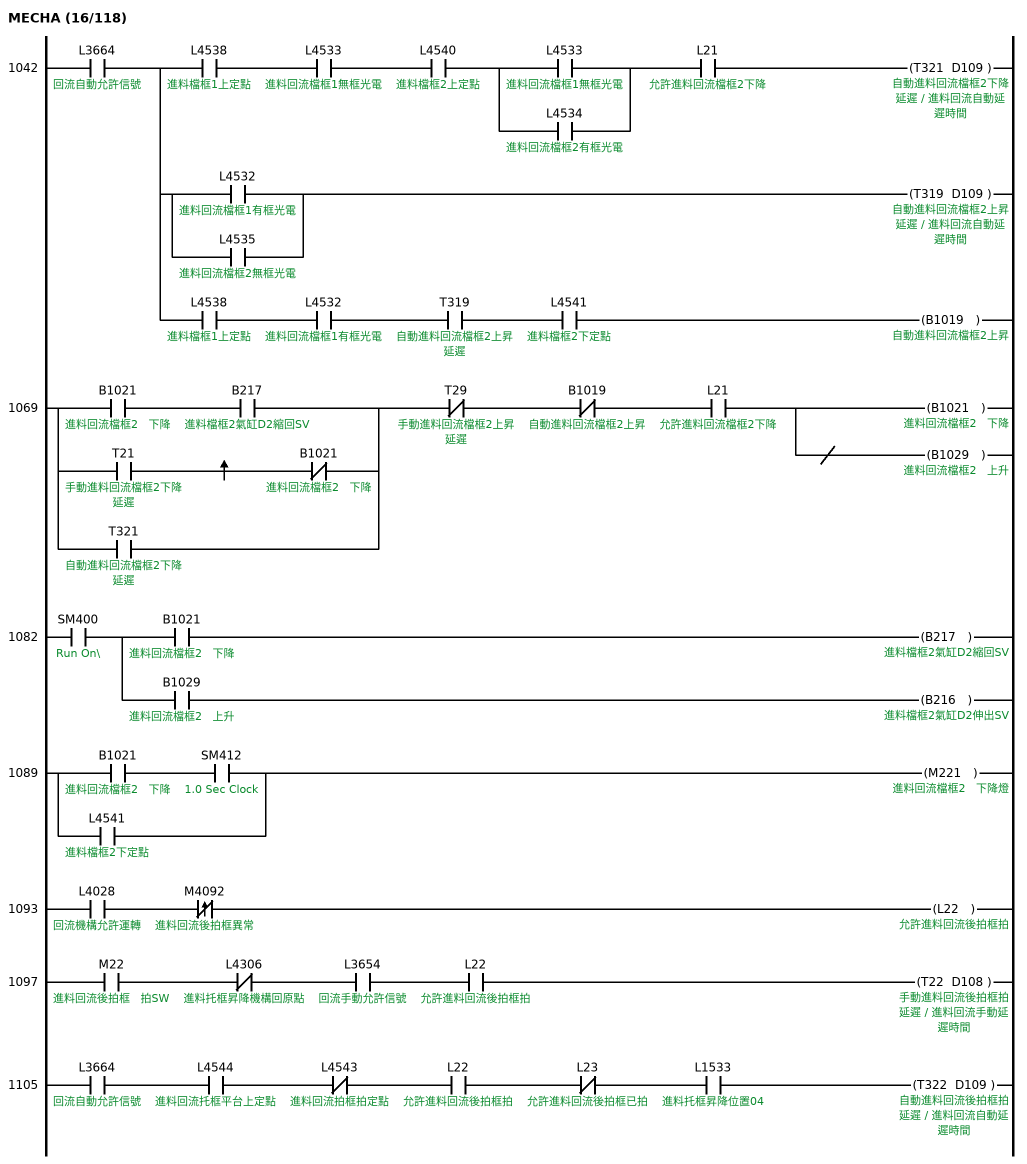
[picture p312: ladder of MECHA, rungs at steps 1042 to 1105]
1042  LD      L3664  ; 回流自動允許信號
      MPS
      AND     L4538  ; 進料檔框1上定點
      AND     L4533  ; 進料回流檔框1無框光電
      AND     L4540  ; 進料檔框2上定點
      LD      L4533  ; 進料回流檔框1無框光電
      OR      L4534  ; 進料回流檔框2有框光電
      ANB
      AND     L21  ; 允許進料回流檔框2下降
      OUT     T321 D109  ; 自動進料回流檔框2下降延遲 / 進料回流自動延遲時間
      MRD
      LD      L4532  ; 進料回流檔框1有框光電
      OR      L4535  ; 進料回流檔框2無框光電
      ANB
      OUT     T319 D109  ; 自動進料回流檔框2上昇延遲 / 進料回流自動延遲時間
      MPP
      AND     L4538  ; 進料檔框1上定點
      AND     L4532  ; 進料回流檔框1有框光電
      AND     T319  ; 自動進料回流檔框2上昇延遲
      AND     L4541  ; 進料檔框2下定點
      OUT     B1019  ; 自動進料回流檔框2上昇
1069  LD      B1021  ; 進料回流檔框2   下降
      AND     B217  ; 進料檔框2氣缸D2縮回SV
      LD      T21  ; 手動進料回流檔框2下降延遲
      MEP
      ANI     B1021  ; 進料回流檔框2   下降
      ORB
      OR      T321  ; 自動進料回流檔框2下降延遲
      ANI     T29  ; 手動進料回流檔框2上昇延遲
      ANI     B1019  ; 自動進料回流檔框2上昇
      AND     L21  ; 允許進料回流檔框2下降
      OUT     B1021  ; 進料回流檔框2   下降
      INV
      OUT     B1029  ; 進料回流檔框2   上升
1082  LD      SM400  ; Run On\
      MPS
      AND     B1021  ; 進料回流檔框2   下降
      OUT     B217  ; 進料檔框2氣缸D2縮回SV
      MPP
      AND     B1029  ; 進料回流檔框2   上升
      OUT     B216  ; 進料檔框2氣缸D2伸出SV
1089  LD      B1021  ; 進料回流檔框2   下降
      AND     SM412  ; 1.0 Sec Clock
      OR      L4541  ; 進料檔框2下定點
      OUT     M221  ; 進料回流檔框2   下降燈
1093  LD      L4028  ; 回流機構允許運轉
      ANDPI   M4092  ; 進料回流後拍框異常
      OUT     L22  ; 允許進料回流後拍框拍
1097  LD      M22  ; 進料回流後拍框   拍SW
      ANI     L4306  ; 進料托框昇降機構回原點
      AND     L3654  ; 回流手動允許信號
      AND     L22  ; 允許進料回流後拍框拍
      OUT     T22 D108  ; 手動進料回流後拍框拍延遲 / 進料回流手動延遲時間
1105  LD      L3664  ; 回流自動允許信號
      AND     L4544  ; 進料回流托框平台上定點
      ANI     L4543  ; 進料回流拍框拍定點
      AND     L22  ; 允許進料回流後拍框拍
      ANI     L23  ; 允許進料回流後拍框已拍
      AND     L1533  ; 進料托框昇降位置04
      OUT     T322 D109  ; 自動進料回流後拍框拍延遲 / 進料回流自動延遲時間
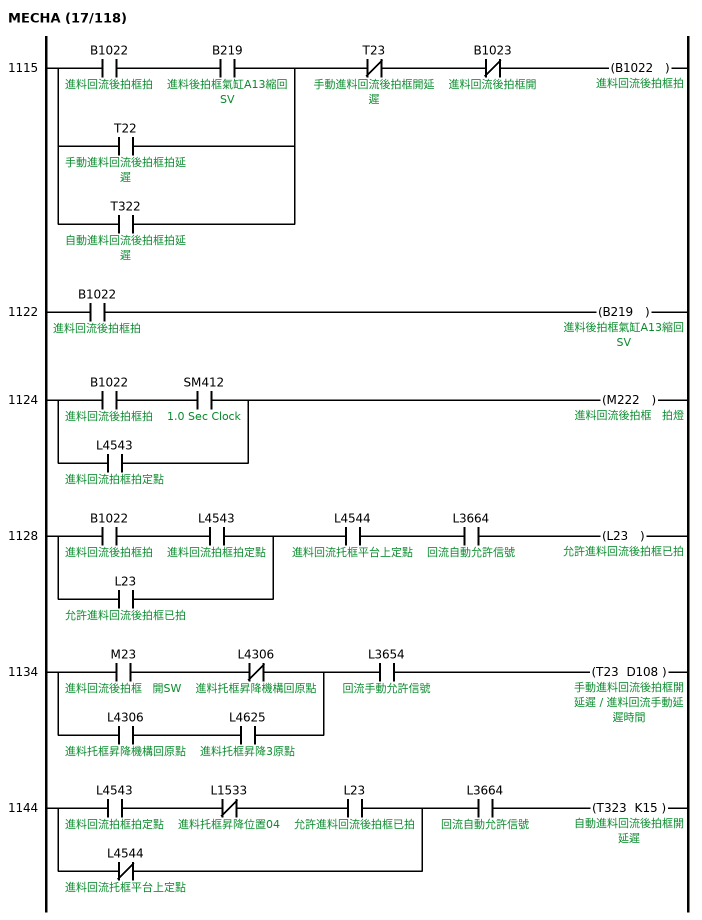
1115  LD      B1022  ; 進料回流後拍框拍
      AND     B219  ; 進料後拍框氣缸A13縮回SV
      OR      T22  ; 手動進料回流後拍框拍延遲
      OR      T322  ; 自動進料回流後拍框拍延遲
      ANI     T23  ; 手動進料回流後拍框開延遲
      ANI     B1023  ; 進料回流後拍框開
      OUT     B1022  ; 進料回流後拍框拍
1122  LD      B1022  ; 進料回流後拍框拍
      OUT     B219  ; 進料後拍框氣缸A13縮回SV
1124  LD      B1022  ; 進料回流後拍框拍
      AND     SM412  ; 1.0 Sec Clock
      OR      L4543  ; 進料回流拍框拍定點
      OUT     M222  ; 進料回流後拍框   拍燈
1128  LD      B1022  ; 進料回流後拍框拍
      AND     L4543  ; 進料回流拍框拍定點
      OR      L23  ; 允許進料回流後拍框已拍
      AND     L4544  ; 進料回流托框平台上定點
      AND     L3664  ; 回流自動允許信號
      OUT     L23  ; 允許進料回流後拍框已拍
1134  LD      M23  ; 進料回流後拍框   開SW
      ANI     L4306  ; 進料托框昇降機構回原點
      LD      L4306  ; 進料托框昇降機構回原點
      AND     L4625  ; 進料托框昇降3原點
      ORB
      AND     L3654  ; 回流手動允許信號
      OUT     T23 D108  ; 手動進料回流後拍框開延遲 / 進料回流手動延遲時間
1144  LD      L4543  ; 進料回流拍框拍定點
      ANI     L1533  ; 進料托框昇降位置04
      AND     L23  ; 允許進料回流後拍框已拍
      ORI     L4544  ; 進料回流托框平台上定點
      AND     L3664  ; 回流自動允許信號
      OUT     T323 K15  ; 自動進料回流後拍框開延遲
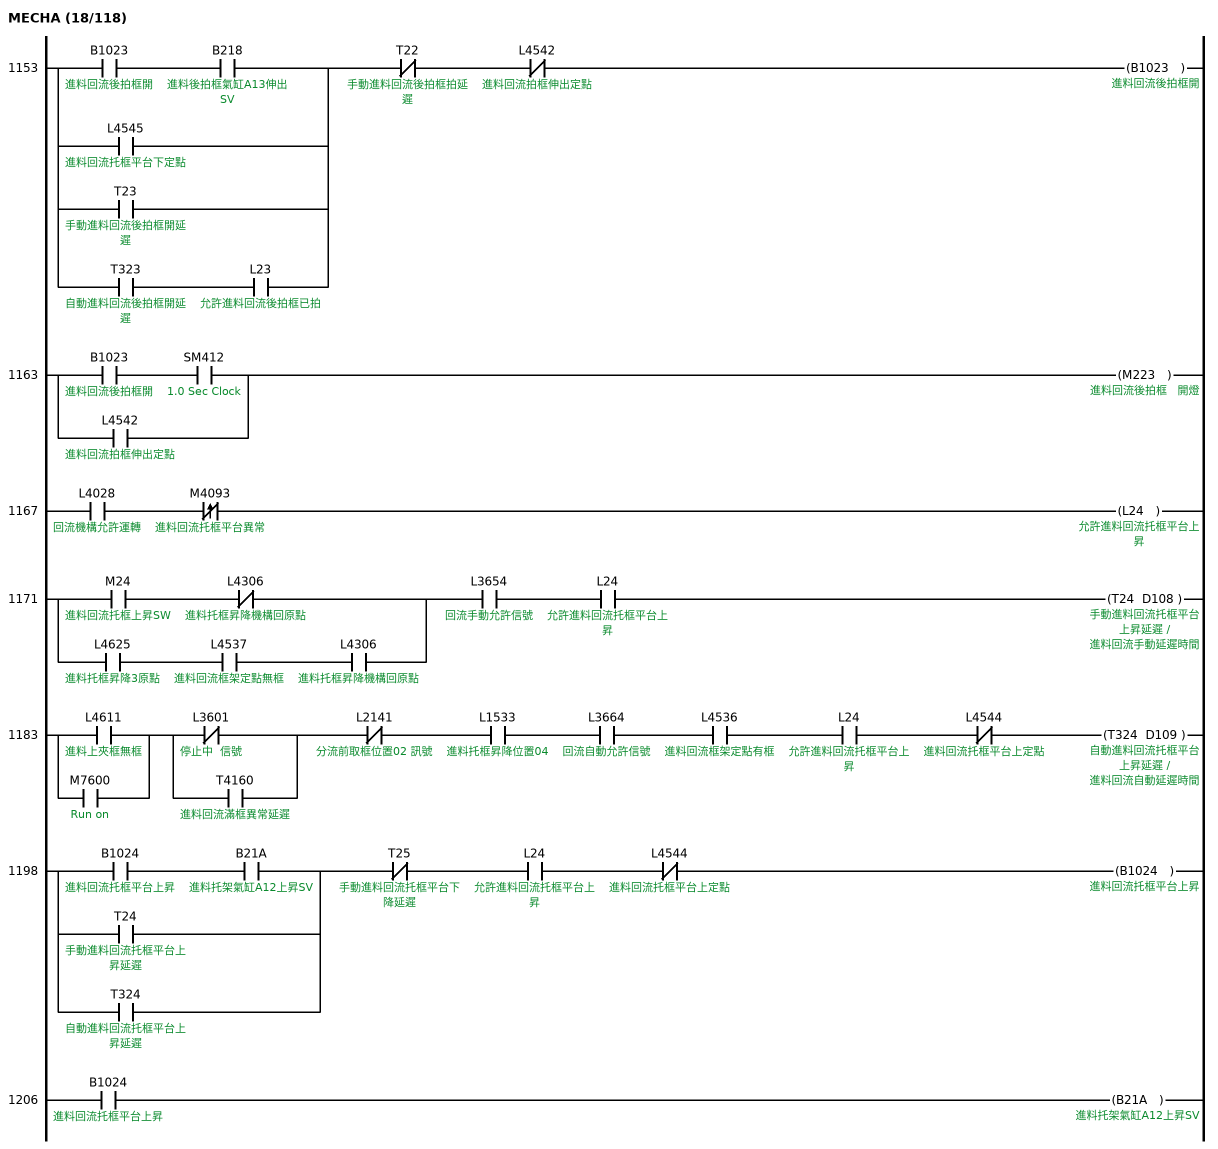
1153  LD      B1023  ; 進料回流後拍框開
      AND     B218  ; 進料後拍框氣缸A13伸出SV
      OR      L4545  ; 進料回流托框平台下定點
      OR      T23  ; 手動進料回流後拍框開延遲
      LD      T323  ; 自動進料回流後拍框開延遲
      AND     L23  ; 允許進料回流後拍框已拍
      ORB
      ANI     T22  ; 手動進料回流後拍框拍延遲
      ANI     L4542  ; 進料回流拍框伸出定點
      OUT     B1023  ; 進料回流後拍框開
1163  LD      B1023  ; 進料回流後拍框開
      AND     SM412  ; 1.0 Sec Clock
      OR      L4542  ; 進料回流拍框伸出定點
      OUT     M223  ; 進料回流後拍框   開燈
1167  LD      L4028  ; 回流機構允許運轉
      ANDPI   M4093  ; 進料回流托框平台異常
      OUT     L24  ; 允許進料回流托框平台上昇
1171  LD      M24  ; 進料回流托框上昇SW
      ANI     L4306  ; 進料托框昇降機構回原點
      LD      L4625  ; 進料托框昇降3原點
      AND     L4537  ; 進料回流框架定點無框
      AND     L4306  ; 進料托框昇降機構回原點
      ORB
      AND     L3654  ; 回流手動允許信號
      AND     L24  ; 允許進料回流托框平台上昇
      OUT     T24 D108  ; 手動進料回流托框平台上昇延遲 / 進料回流手動延遲時間
1183  LD      L4611  ; 進料上夾框無框
      OR      M7600  ; Run on
      LDI     L3601  ; 停止中  信號
      OR      T4160  ; 進料回流滿框異常延遲
      ANB
      ANI     L2141  ; 分流前取框位置02 訊號
      AND     L1533  ; 進料托框昇降位置04
      AND     L3664  ; 回流自動允許信號
      AND     L4536  ; 進料回流框架定點有框
      AND     L24  ; 允許進料回流托框平台上昇
      ANI     L4544  ; 進料回流托框平台上定點
      OUT     T324 D109  ; 自動進料回流托框平台上昇延遲 / 進料回流自動延遲時間
1198  LD      B1024  ; 進料回流托框平台上昇
      AND     B21A  ; 進料托架氣缸A12上昇SV
      OR      T24  ; 手動進料回流托框平台上昇延遲
      OR      T324  ; 自動進料回流托框平台上昇延遲
      ANI     T25  ; 手動進料回流托框平台下降延遲
      AND     L24  ; 允許進料回流托框平台上昇
      ANI     L4544  ; 進料回流托框平台上定點
      OUT     B1024  ; 進料回流托框平台上昇
1206  LD      B1024  ; 進料回流托框平台上昇
      OUT     B21A  ; 進料托架氣缸A12上昇SV
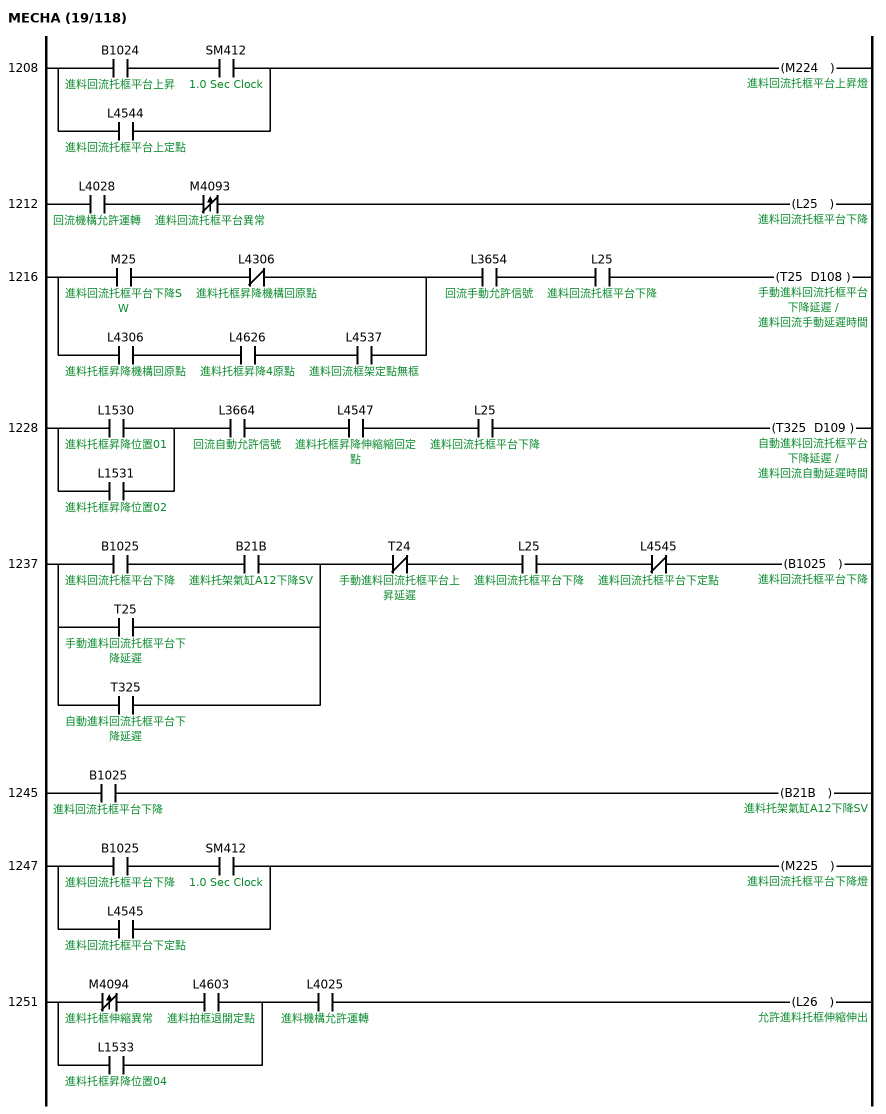
1208  LD      B1024  ; 進料回流托框平台上昇
      AND     SM412  ; 1.0 Sec Clock
      OR      L4544  ; 進料回流托框平台上定點
      OUT     M224  ; 進料回流托框平台上昇燈
1212  LD      L4028  ; 回流機構允許運轉
      ANDPI   M4093  ; 進料回流托框平台異常
      OUT     L25  ; 進料回流托框平台下降
1216  LD      M25  ; 進料回流托框平台下降SW
      ANI     L4306  ; 進料托框昇降機構回原點
      LD      L4306  ; 進料托框昇降機構回原點
      AND     L4626  ; 進料托框昇降4原點
      AND     L4537  ; 進料回流框架定點無框
      ORB
      AND     L3654  ; 回流手動允許信號
      AND     L25  ; 進料回流托框平台下降
      OUT     T25 D108  ; 手動進料回流托框平台下降延遲 / 進料回流手動延遲時間
1228  LD      L1530  ; 進料托框昇降位置01
      OR      L1531  ; 進料托框昇降位置02
      AND     L3664  ; 回流自動允許信號
      AND     L4547  ; 進料托框昇降伸縮縮回定點
      AND     L25  ; 進料回流托框平台下降
      OUT     T325 D109  ; 自動進料回流托框平台下降延遲 / 進料回流自動延遲時間
1237  LD      B1025  ; 進料回流托框平台下降
      AND     B21B  ; 進料托架氣缸A12下降SV
      OR      T25  ; 手動進料回流托框平台下降延遲
      OR      T325  ; 自動進料回流托框平台下降延遲
      ANI     T24  ; 手動進料回流托框平台上昇延遲
      AND     L25  ; 進料回流托框平台下降
      ANI     L4545  ; 進料回流托框平台下定點
      OUT     B1025  ; 進料回流托框平台下降
1245  LD      B1025  ; 進料回流托框平台下降
      OUT     B21B  ; 進料托架氣缸A12下降SV
1247  LD      B1025  ; 進料回流托框平台下降
      AND     SM412  ; 1.0 Sec Clock
      OR      L4545  ; 進料回流托框平台下定點
      OUT     M225  ; 進料回流托框平台下降燈
1251  LDPI    M4094  ; 進料托框伸縮異常
      AND     L4603  ; 進料拍框退開定點
      OR      L1533  ; 進料托框昇降位置04
      AND     L4025  ; 進料機構允許運轉
      OUT     L26  ; 允許進料托框伸縮伸出
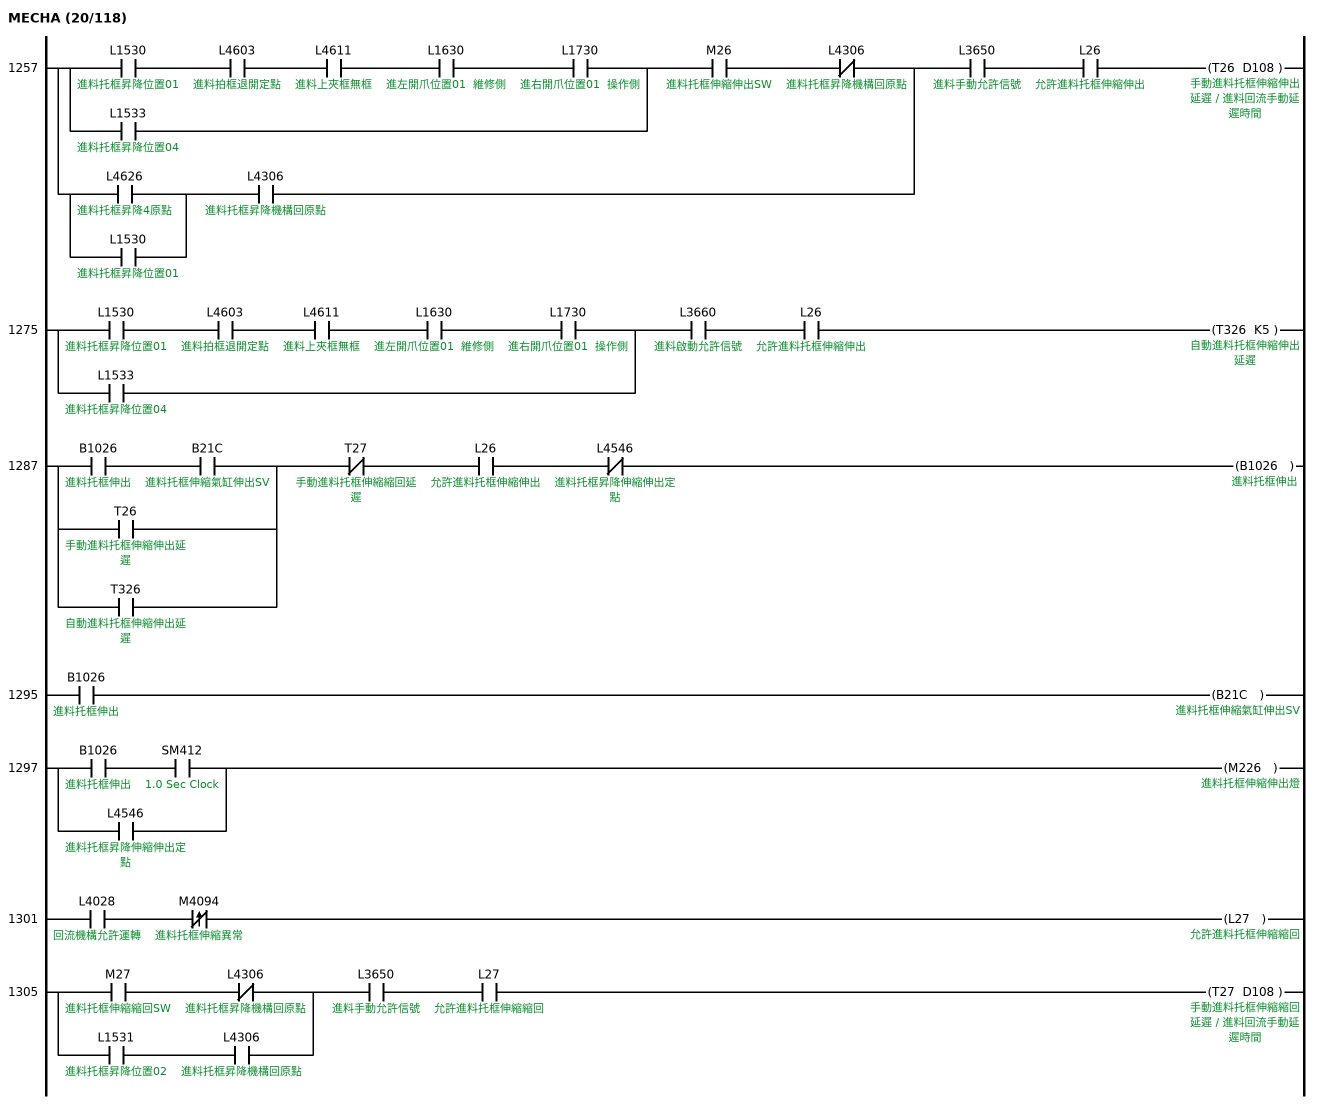
1257  LD      L1530  ; 進料托框昇降位置01
      AND     L4603  ; 進料拍框退開定點
      AND     L4611  ; 進料上夾框無框
      AND     L1630  ; 進左開爪位置01  維修側
      AND     L1730  ; 進右開爪位置01  操作側
      OR      L1533  ; 進料托框昇降位置04
      AND     M26  ; 進料托框伸縮伸出SW
      ANI     L4306  ; 進料托框昇降機構回原點
      LD      L4626  ; 進料托框昇降4原點
      OR      L1530  ; 進料托框昇降位置01
      AND     L4306  ; 進料托框昇降機構回原點
      ORB
      AND     L3650  ; 進料手動允許信號
      AND     L26  ; 允許進料托框伸縮伸出
      OUT     T26 D108  ; 手動進料托框伸縮伸出延遲 / 進料回流手動延遲時間
1275  LD      L1530  ; 進料托框昇降位置01
      AND     L4603  ; 進料拍框退開定點
      AND     L4611  ; 進料上夾框無框
      AND     L1630  ; 進左開爪位置01  維修側
      AND     L1730  ; 進右開爪位置01  操作側
      OR      L1533  ; 進料托框昇降位置04
      AND     L3660  ; 進料啟動允許信號
      AND     L26  ; 允許進料托框伸縮伸出
      OUT     T326 K5  ; 自動進料托框伸縮伸出延遲
1287  LD      B1026  ; 進料托框伸出
      AND     B21C  ; 進料托框伸縮氣缸伸出SV
      OR      T26  ; 手動進料托框伸縮伸出延遲
      OR      T326  ; 自動進料托框伸縮伸出延遲
      ANI     T27  ; 手動進料托框伸縮縮回延遲
      AND     L26  ; 允許進料托框伸縮伸出
      ANI     L4546  ; 進料托框昇降伸縮伸出定點
      OUT     B1026  ; 進料托框伸出
1295  LD      B1026  ; 進料托框伸出
      OUT     B21C  ; 進料托框伸縮氣缸伸出SV
1297  LD      B1026  ; 進料托框伸出
      AND     SM412  ; 1.0 Sec Clock
      OR      L4546  ; 進料托框昇降伸縮伸出定點
      OUT     M226  ; 進料托框伸縮伸出燈
1301  LD      L4028  ; 回流機構允許運轉
      ANDPI   M4094  ; 進料托框伸縮異常
      OUT     L27  ; 允許進料托框伸縮縮回
1305  LD      M27  ; 進料托框伸縮縮回SW
      ANI     L4306  ; 進料托框昇降機構回原點
      LD      L1531  ; 進料托框昇降位置02
      AND     L4306  ; 進料托框昇降機構回原點
      ORB
      AND     L3650  ; 進料手動允許信號
      AND     L27  ; 允許進料托框伸縮縮回
      OUT     T27 D108  ; 手動進料托框伸縮縮回延遲 / 進料回流手動延遲時間
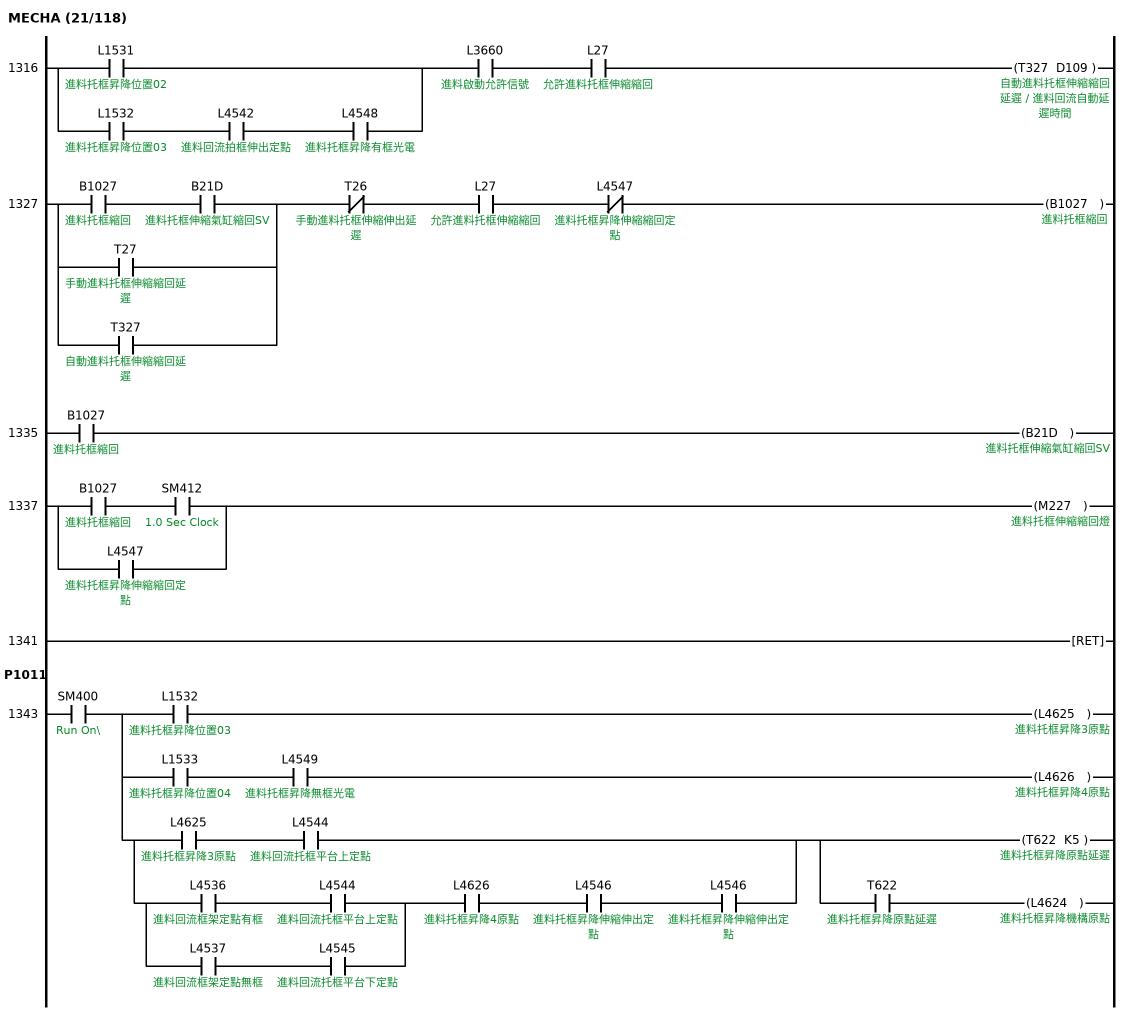
1316  LD      L1531  ; 進料托框昇降位置02
      LD      L1532  ; 進料托框昇降位置03
      AND     L4542  ; 進料回流拍框伸出定點
      AND     L4548  ; 進料托框昇降有框光電
      ORB
      AND     L3660  ; 進料啟動允許信號
      AND     L27  ; 允許進料托框伸縮縮回
      OUT     T327 D109  ; 自動進料托框伸縮縮回延遲 / 進料回流自動延遲時間
1327  LD      B1027  ; 進料托框縮回
      AND     B21D  ; 進料托框伸縮氣缸縮回SV
      OR      T27  ; 手動進料托框伸縮縮回延遲
      OR      T327  ; 自動進料托框伸縮縮回延遲
      ANI     T26  ; 手動進料托框伸縮伸出延遲
      AND     L27  ; 允許進料托框伸縮縮回
      ANI     L4547  ; 進料托框昇降伸縮縮回定點
      OUT     B1027  ; 進料托框縮回
1335  LD      B1027  ; 進料托框縮回
      OUT     B21D  ; 進料托框伸縮氣缸縮回SV
1337  LD      B1027  ; 進料托框縮回
      AND     SM412  ; 1.0 Sec Clock
      OR      L4547  ; 進料托框昇降伸縮縮回定點
      OUT     M227  ; 進料托框伸縮縮回燈
1341  RET
      P1011
1343  LD      SM400  ; Run On\
      MPS
      AND     L1532  ; 進料托框昇降位置03
      OUT     L4625  ; 進料托框昇降3原點
      MRD
      AND     L1533  ; 進料托框昇降位置04
      AND     L4549  ; 進料托框昇降無框光電
      OUT     L4626  ; 進料托框昇降4原點
      MPP
      LD      L4625  ; 進料托框昇降3原點
      AND     L4544  ; 進料回流托框平台上定點
      LD      L4536  ; 進料回流框架定點有框
      AND     L4544  ; 進料回流托框平台上定點
      LD      L4537  ; 進料回流框架定點無框
      AND     L4545  ; 進料回流托框平台下定點
      ORB
      AND     L4626  ; 進料托框昇降4原點
      AND     L4546  ; 進料托框昇降伸縮伸出定點
      AND     L4546  ; 進料托框昇降伸縮伸出定點
      ORB
      ANB
      OUT     T622 K5  ; 進料托框昇降原點延遲
      AND     T622  ; 進料托框昇降原點延遲
      OUT     L4624  ; 進料托框昇降機構原點
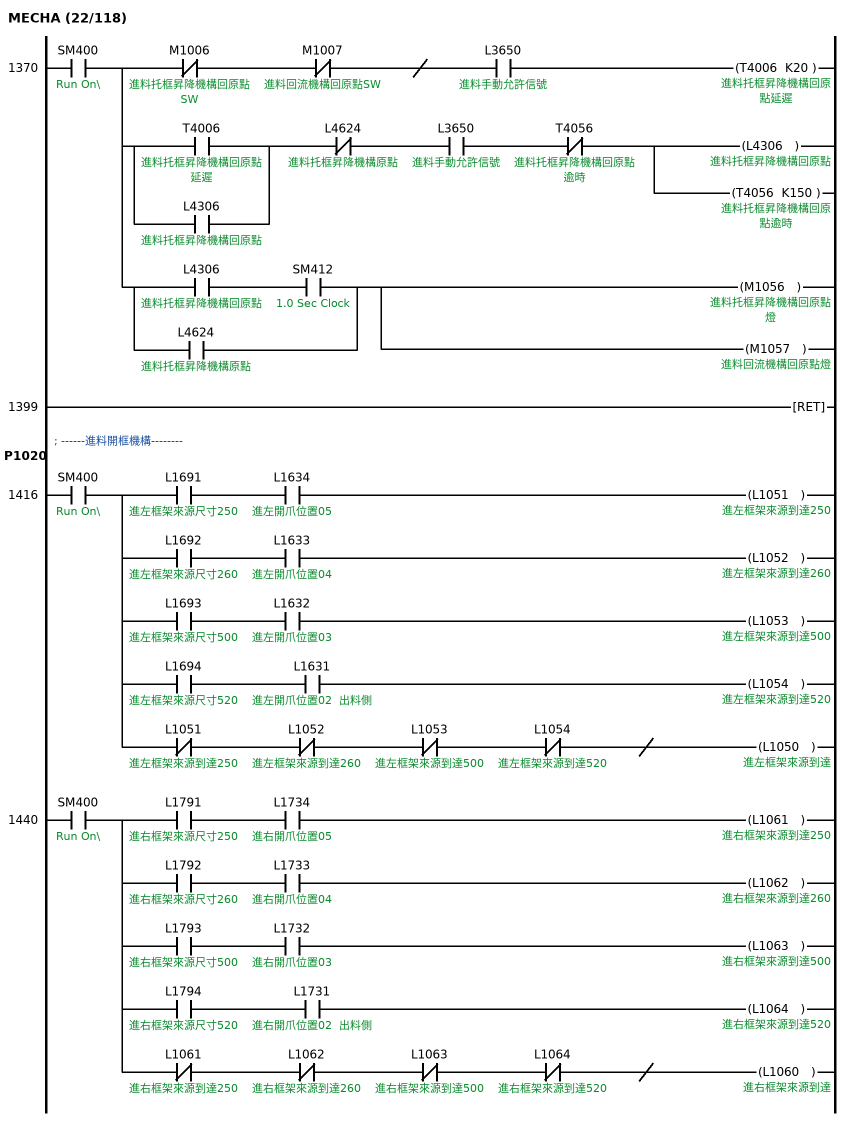
1370  LD      SM400  ; Run On\
      MPS
      ANI     M1006  ; 進料托框昇降機構回原點SW
      ANI     M1007  ; 進料回流機構回原點SW
      INV
      AND     L3650  ; 進料手動允許信號
      OUT     T4006 K20  ; 進料托框昇降機構回原點延遲
      MRD
      LD      T4006  ; 進料托框昇降機構回原點延遲
      OR      L4306  ; 進料托框昇降機構回原點
      ANB
      ANI     L4624  ; 進料托框昇降機構原點
      AND     L3650  ; 進料手動允許信號
      ANI     T4056  ; 進料托框昇降機構回原點逾時
      OUT     L4306  ; 進料托框昇降機構回原點
      OUT     T4056 K150  ; 進料托框昇降機構回原點逾時
      MPP
      LD      L4306  ; 進料托框昇降機構回原點
      AND     SM412  ; 1.0 Sec Clock
      OR      L4624  ; 進料托框昇降機構原點
      ANB
      OUT     M1056  ; 進料托框昇降機構回原點燈
      OUT     M1057  ; 進料回流機構回原點燈
1399  RET
; ------進料開框機構--------
      P1020
1416  LD      SM400  ; Run On\
      MPS
      AND     L1691  ; 進左框架來源尺寸250
      AND     L1634  ; 進左開爪位置05
      OUT     L1051  ; 進左框架來源到達250
      MRD
      AND     L1692  ; 進左框架來源尺寸260
      AND     L1633  ; 進左開爪位置04
      OUT     L1052  ; 進左框架來源到達260
      MRD
      AND     L1693  ; 進左框架來源尺寸500
      AND     L1632  ; 進左開爪位置03
      OUT     L1053  ; 進左框架來源到達500
      MRD
      AND     L1694  ; 進左框架來源尺寸520
      AND     L1631  ; 進左開爪位置02  出料側
      OUT     L1054  ; 進左框架來源到達520
      MPP
      ANI     L1051  ; 進左框架來源到達250
      ANI     L1052  ; 進左框架來源到達260
      ANI     L1053  ; 進左框架來源到達500
      ANI     L1054  ; 進左框架來源到達520
      INV
      OUT     L1050  ; 進左框架來源到達
1440  LD      SM400  ; Run On\
      MPS
      AND     L1791  ; 進右框架來源尺寸250
      AND     L1734  ; 進右開爪位置05
      OUT     L1061  ; 進右框架來源到達250
      MRD
      AND     L1792  ; 進右框架來源尺寸260
      AND     L1733  ; 進右開爪位置04
      OUT     L1062  ; 進右框架來源到達260
      MRD
      AND     L1793  ; 進右框架來源尺寸500
      AND     L1732  ; 進右開爪位置03
      OUT     L1063  ; 進右框架來源到達500
      MRD
      AND     L1794  ; 進右框架來源尺寸520
      AND     L1731  ; 進右開爪位置02  出料側
      OUT     L1064  ; 進右框架來源到達520
      MPP
      ANI     L1061  ; 進右框架來源到達250
      ANI     L1062  ; 進右框架來源到達260
      ANI     L1063  ; 進右框架來源到達500
      ANI     L1064  ; 進右框架來源到達520
      INV
      OUT     L1060  ; 進右框架來源到達
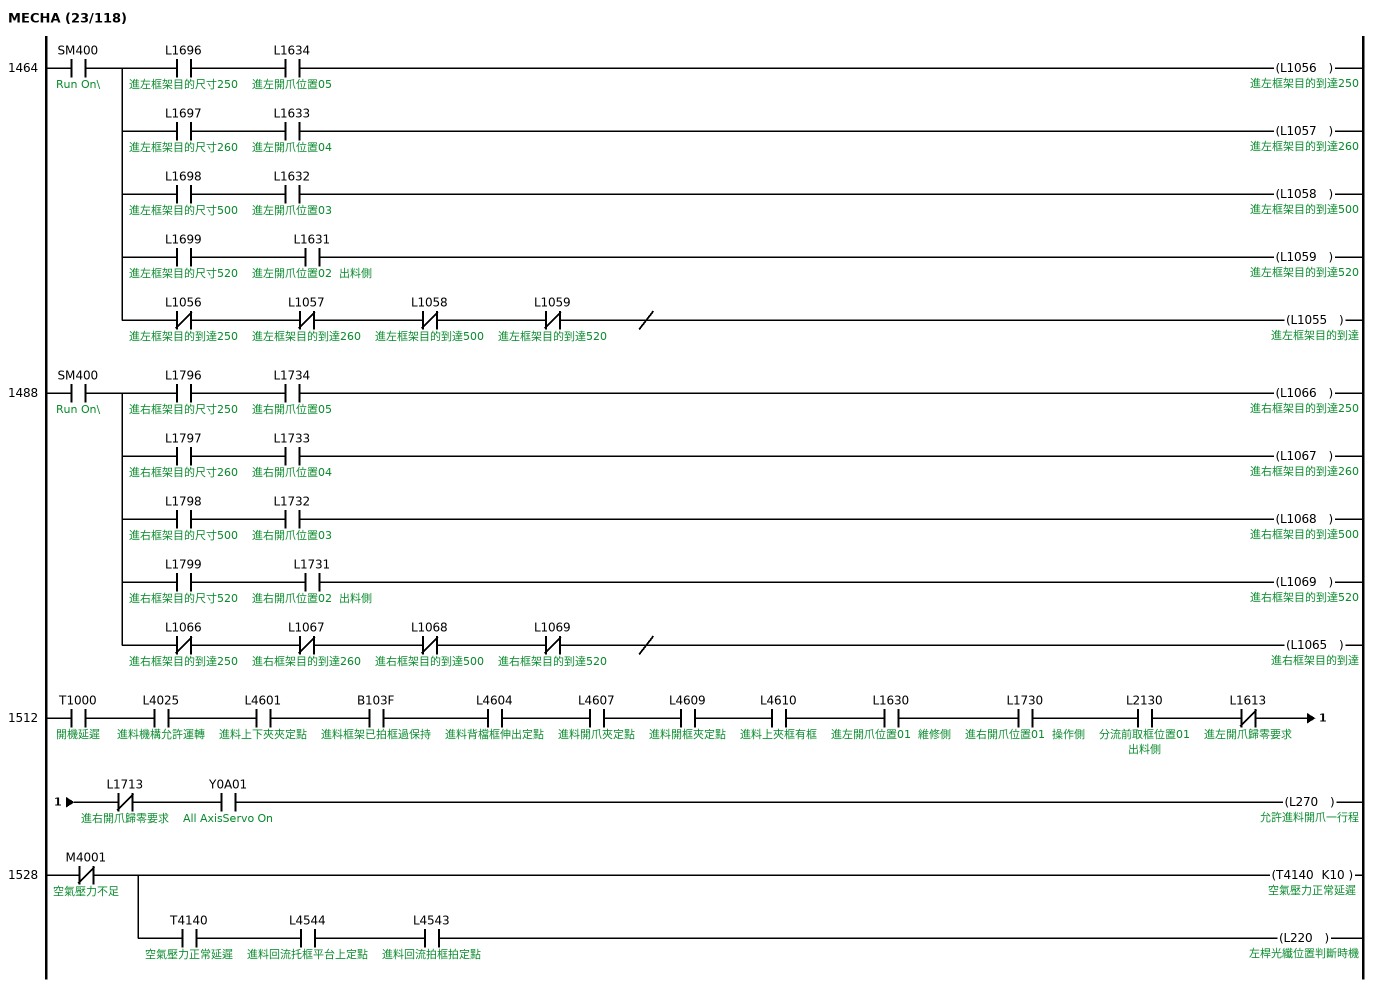
1464  LD      SM400  ; Run On\
      MPS
      AND     L1696  ; 進左框架目的尺寸250
      AND     L1634  ; 進左開爪位置05
      OUT     L1056  ; 進左框架目的到達250
      MRD
      AND     L1697  ; 進左框架目的尺寸260
      AND     L1633  ; 進左開爪位置04
      OUT     L1057  ; 進左框架目的到達260
      MRD
      AND     L1698  ; 進左框架目的尺寸500
      AND     L1632  ; 進左開爪位置03
      OUT     L1058  ; 進左框架目的到達500
      MRD
      AND     L1699  ; 進左框架目的尺寸520
      AND     L1631  ; 進左開爪位置02  出料側
      OUT     L1059  ; 進左框架目的到達520
      MPP
      ANI     L1056  ; 進左框架目的到達250
      ANI     L1057  ; 進左框架目的到達260
      ANI     L1058  ; 進左框架目的到達500
      ANI     L1059  ; 進左框架目的到達520
      INV
      OUT     L1055  ; 進左框架目的到達
1488  LD      SM400  ; Run On\
      MPS
      AND     L1796  ; 進右框架目的尺寸250
      AND     L1734  ; 進右開爪位置05
      OUT     L1066  ; 進右框架目的到達250
      MRD
      AND     L1797  ; 進右框架目的尺寸260
      AND     L1733  ; 進右開爪位置04
      OUT     L1067  ; 進右框架目的到達260
      MRD
      AND     L1798  ; 進右框架目的尺寸500
      AND     L1732  ; 進右開爪位置03
      OUT     L1068  ; 進右框架目的到達500
      MRD
      AND     L1799  ; 進右框架目的尺寸520
      AND     L1731  ; 進右開爪位置02  出料側
      OUT     L1069  ; 進右框架目的到達520
      MPP
      ANI     L1066  ; 進右框架目的到達250
      ANI     L1067  ; 進右框架目的到達260
      ANI     L1068  ; 進右框架目的到達500
      ANI     L1069  ; 進右框架目的到達520
      INV
      OUT     L1065  ; 進右框架目的到達
1512  LD      T1000  ; 開機延遲
      AND     L4025  ; 進料機構允許運轉
      AND     L4601  ; 進料上下夾夾定點
      AND     B103F  ; 進料框架已拍框過保持
      AND     L4604  ; 進料背檔框伸出定點
      AND     L4607  ; 進料開爪夾定點
      AND     L4609  ; 進料開框夾定點
      AND     L4610  ; 進料上夾框有框
      AND     L1630  ; 進左開爪位置01  維修側
      AND     L1730  ; 進右開爪位置01  操作側
      AND     L2130  ; 分流前取框位置01  出料側
      ANI     L1613  ; 進左開爪歸零要求
      ANI     L1713  ; 進右開爪歸零要求
      AND     Y0A01  ; All AxisServo On
      OUT     L270  ; 允許進料開爪一行程
1528  LDI     M4001  ; 空氣壓力不足
      OUT     T4140 K10  ; 空氣壓力正常延遲
      AND     T4140  ; 空氣壓力正常延遲
      AND     L4544  ; 進料回流托框平台上定點
      AND     L4543  ; 進料回流拍框拍定點
      OUT     L220  ; 左桿光纖位置判斷時機
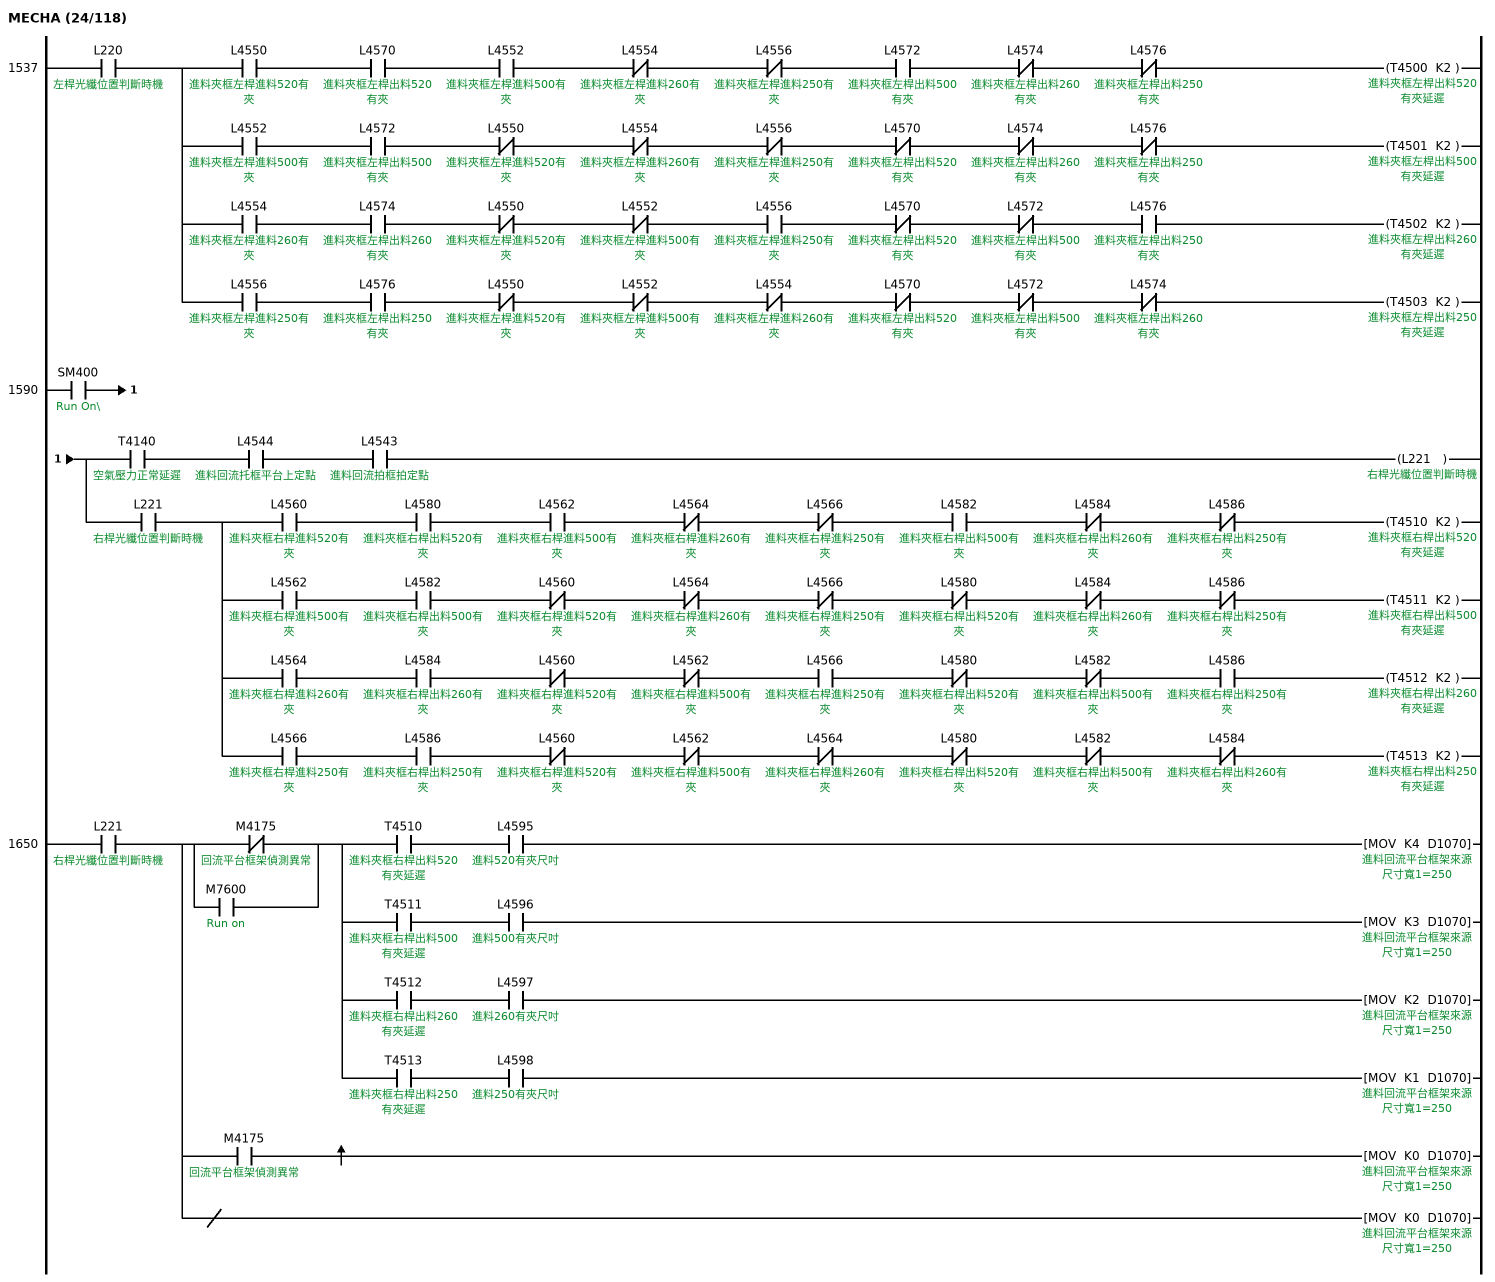
1537  LD      L220  ; 左桿光纖位置判斷時機
      MPS
      AND     L4550  ; 進料夾框左桿進料520有夾
      AND     L4570  ; 進料夾框左桿出料520 有夾
      AND     L4552  ; 進料夾框左桿進料500有夾
      ANI     L4554  ; 進料夾框左桿進料260有夾
      ANI     L4556  ; 進料夾框左桿進料250有夾
      AND     L4572  ; 進料夾框左桿出料500 有夾
      ANI     L4574  ; 進料夾框左桿出料260 有夾
      ANI     L4576  ; 進料夾框左桿出料250 有夾
      OUT     T4500 K2  ; 進料夾框左桿出料520 有夾延遲
      MRD
      AND     L4552  ; 進料夾框左桿進料500有夾
      AND     L4572  ; 進料夾框左桿出料500 有夾
      ANI     L4550  ; 進料夾框左桿進料520有夾
      ANI     L4554  ; 進料夾框左桿進料260有夾
      ANI     L4556  ; 進料夾框左桿進料250有夾
      ANI     L4570  ; 進料夾框左桿出料520 有夾
      ANI     L4574  ; 進料夾框左桿出料260 有夾
      ANI     L4576  ; 進料夾框左桿出料250 有夾
      OUT     T4501 K2  ; 進料夾框左桿出料500 有夾延遲
      MRD
      AND     L4554  ; 進料夾框左桿進料260有夾
      AND     L4574  ; 進料夾框左桿出料260 有夾
      ANI     L4550  ; 進料夾框左桿進料520有夾
      ANI     L4552  ; 進料夾框左桿進料500有夾
      AND     L4556  ; 進料夾框左桿進料250有夾
      ANI     L4570  ; 進料夾框左桿出料520 有夾
      ANI     L4572  ; 進料夾框左桿出料500 有夾
      AND     L4576  ; 進料夾框左桿出料250 有夾
      OUT     T4502 K2  ; 進料夾框左桿出料260 有夾延遲
      MPP
      AND     L4556  ; 進料夾框左桿進料250有夾
      AND     L4576  ; 進料夾框左桿出料250 有夾
      ANI     L4550  ; 進料夾框左桿進料520有夾
      ANI     L4552  ; 進料夾框左桿進料500有夾
      ANI     L4554  ; 進料夾框左桿進料260有夾
      ANI     L4570  ; 進料夾框左桿出料520 有夾
      ANI     L4572  ; 進料夾框左桿出料500 有夾
      ANI     L4574  ; 進料夾框左桿出料260 有夾
      OUT     T4503 K2  ; 進料夾框左桿出料250 有夾延遲
1590  LD      SM400  ; Run On\
      MPS
      AND     T4140  ; 空氣壓力正常延遲
      AND     L4544  ; 進料回流托框平台上定點
      AND     L4543  ; 進料回流拍框拍定點
      OUT     L221  ; 右桿光纖位置判斷時機
      MPP
      AND     L221  ; 右桿光纖位置判斷時機
      MPS
      AND     L4560  ; 進料夾框右桿進料520有夾
      AND     L4580  ; 進料夾框右桿出料520有夾
      AND     L4562  ; 進料夾框右桿進料500有夾
      ANI     L4564  ; 進料夾框右桿進料260有夾
      ANI     L4566  ; 進料夾框右桿進料250有夾
      AND     L4582  ; 進料夾框右桿出料500有夾
      ANI     L4584  ; 進料夾框右桿出料260有夾
      ANI     L4586  ; 進料夾框右桿出料250有夾
      OUT     T4510 K2  ; 進料夾框右桿出料520 有夾延遲
      MRD
      AND     L4562  ; 進料夾框右桿進料500有夾
      AND     L4582  ; 進料夾框右桿出料500有夾
      ANI     L4560  ; 進料夾框右桿進料520有夾
      ANI     L4564  ; 進料夾框右桿進料260有夾
      ANI     L4566  ; 進料夾框右桿進料250有夾
      ANI     L4580  ; 進料夾框右桿出料520有夾
      ANI     L4584  ; 進料夾框右桿出料260有夾
      ANI     L4586  ; 進料夾框右桿出料250有夾
      OUT     T4511 K2  ; 進料夾框右桿出料500 有夾延遲
      MRD
      AND     L4564  ; 進料夾框右桿進料260有夾
      AND     L4584  ; 進料夾框右桿出料260有夾
      ANI     L4560  ; 進料夾框右桿進料520有夾
      ANI     L4562  ; 進料夾框右桿進料500有夾
      AND     L4566  ; 進料夾框右桿進料250有夾
      ANI     L4580  ; 進料夾框右桿出料520有夾
      ANI     L4582  ; 進料夾框右桿出料500有夾
      AND     L4586  ; 進料夾框右桿出料250有夾
      OUT     T4512 K2  ; 進料夾框右桿出料260 有夾延遲
      MPP
      AND     L4566  ; 進料夾框右桿進料250有夾
      AND     L4586  ; 進料夾框右桿出料250有夾
      ANI     L4560  ; 進料夾框右桿進料520有夾
      ANI     L4562  ; 進料夾框右桿進料500有夾
      ANI     L4564  ; 進料夾框右桿進料260有夾
      ANI     L4580  ; 進料夾框右桿出料520有夾
      ANI     L4582  ; 進料夾框右桿出料500有夾
      ANI     L4584  ; 進料夾框右桿出料260有夾
      OUT     T4513 K2  ; 進料夾框右桿出料250 有夾延遲
1650  LD      L221  ; 右桿光纖位置判斷時機
      MPS
      LDI     M4175  ; 回流平台框架偵測異常
      OR      M7600  ; Run on
      ANB
      MPS
      AND     T4510  ; 進料夾框右桿出料520 有夾延遲
      AND     L4595  ; 進料520有夾尺吋
      MOV     K4 D1070  ; 進料回流平台框架來源尺寸寬1=250
      MRD
      AND     T4511  ; 進料夾框右桿出料500 有夾延遲
      AND     L4596  ; 進料500有夾尺吋
      MOV     K3 D1070
      MRD
      AND     T4512  ; 進料夾框右桿出料260 有夾延遲
      AND     L4597  ; 進料260有夾尺吋
      MOV     K2 D1070
      MPP
      AND     T4513  ; 進料夾框右桿出料250 有夾延遲
      AND     L4598  ; 進料250有夾尺吋
      MOV     K1 D1070
      MRD
      AND     M4175  ; 回流平台框架偵測異常
      MEP
      MOV     K0 D1070
      MPP
      INV
      MOV     K0 D1070
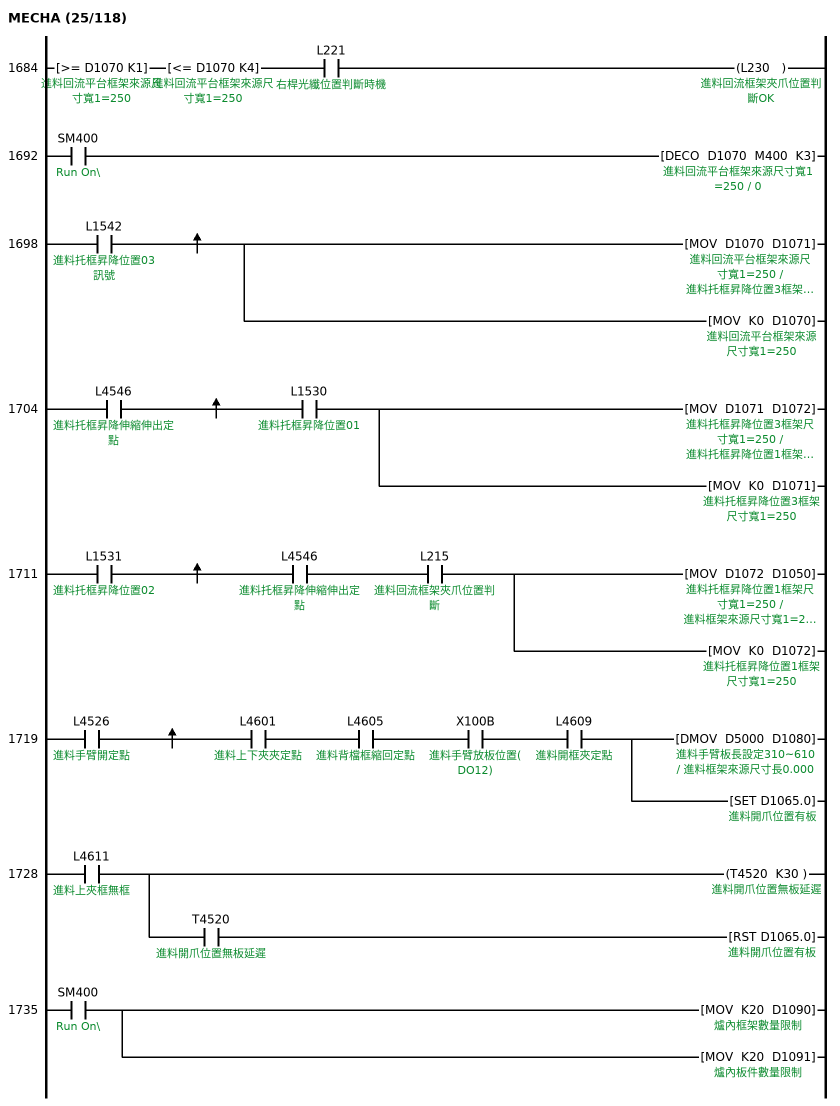
1684  LD>=    D1070 K1  ; 進料回流平台框架來源尺寸寬1=250
      AND<=   D1070 K4  ; 進料回流平台框架來源尺寸寬1=250
      AND     L221  ; 右桿光纖位置判斷時機
      OUT     L230  ; 進料回流框架夾爪位置判斷OK
1692  LD      SM400  ; Run On\
      DECO    D1070 M400 K3  ; 0
1698  LD      L1542  ; 進料托框昇降位置03 訊號
      MEP
      MOV     D1070 D1071  ; 進料托框昇降位置3框架尺寸寬1=250
      MOV     K0 D1070
1704  LD      L4546  ; 進料托框昇降伸縮伸出定點
      MEP
      AND     L1530  ; 進料托框昇降位置01
      MOV     D1071 D1072  ; 進料托框昇降位置1框架尺寸寬1=250
      MOV     K0 D1071
1711  LD      L1531  ; 進料托框昇降位置02
      MEP
      AND     L4546  ; 進料托框昇降伸縮伸出定點
      AND     L215  ; 進料回流框架夾爪位置判斷
      MOV     D1072 D1050  ; 進料框架來源尺寸寬1=250
      MOV     K0 D1072
1719  LD      L4526  ; 進料手臂開定點
      MEP
      AND     L4601  ; 進料上下夾夾定點
      AND     L4605  ; 進料背檔框縮回定點
      AND     X100B  ; 進料手臂放板位置(DO12)
      AND     L4609  ; 進料開框夾定點
      DMOV    D5000 D1080  ; 進料手臂板長設定310~610 / 進料框架來源尺寸長0.000
      SET     D1065.0  ; 進料開爪位置有板
1728  LD      L4611  ; 進料上夾框無框
      OUT     T4520 K30  ; 進料開爪位置無板延遲
      AND     T4520  ; 進料開爪位置無板延遲
      RST     D1065.0  ; 進料開爪位置有板
1735  LD      SM400  ; Run On\
      MOV     K20 D1090  ; 爐內框架數量限制
      MOV     K20 D1091  ; 爐內板件數量限制
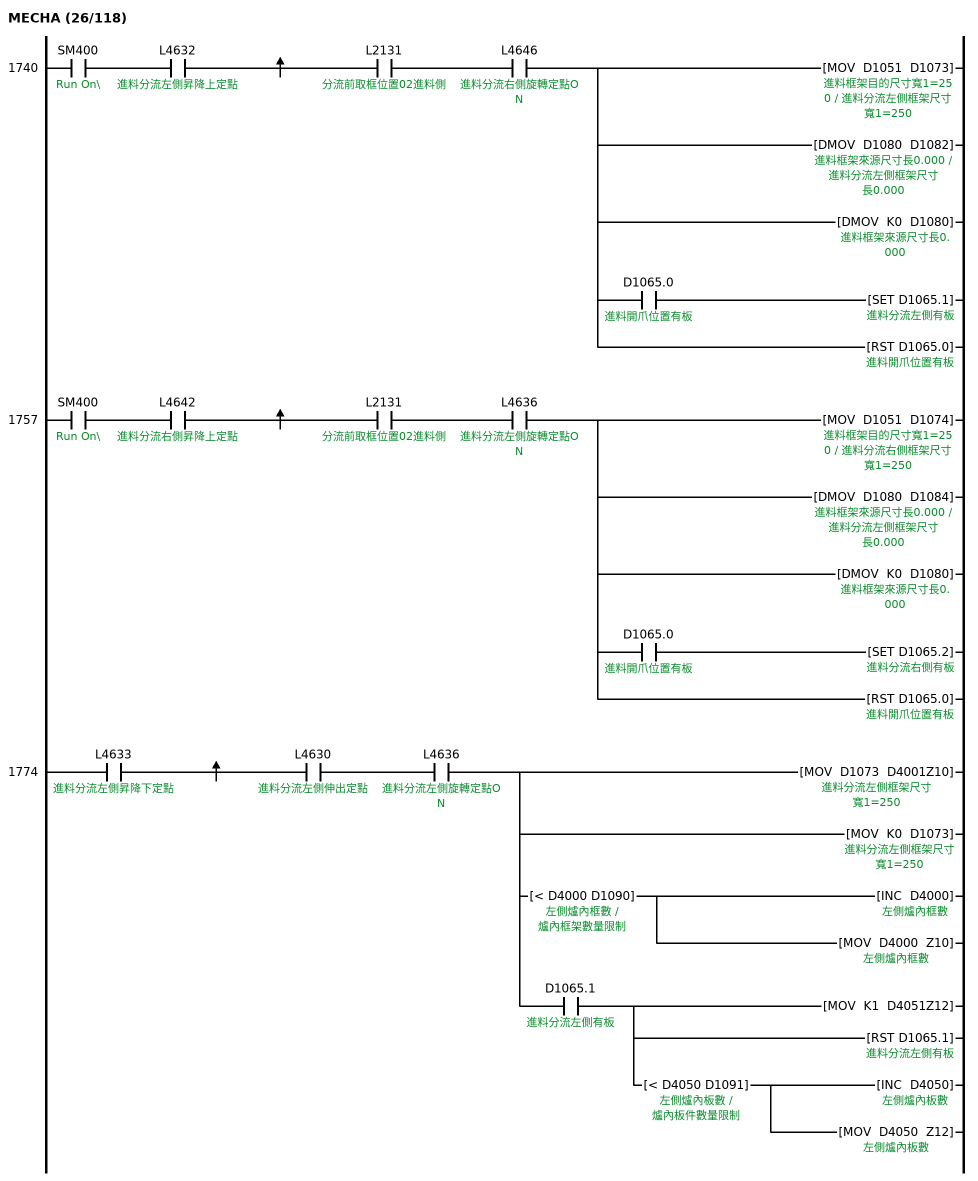
1740  LD      SM400  ; Run On\
      AND     L4632  ; 進料分流左側昇降上定點
      MEP
      AND     L2131  ; 分流前取框位置02進料側
      AND     L4646  ; 進料分流右側旋轉定點ON
      MOV     D1051 D1073  ; 進料框架目的尺寸寬1=250 / 進料分流左側框架尺寸    寬1=250
      DMOV    D1080 D1082  ; 進料分流左側框架尺寸    長0.000
      DMOV    K0 D1080
      MPS
      AND     D1065.0  ; 進料開爪位置有板
      SET     D1065.1  ; 進料分流左側有板
      MPP
      RST     D1065.0  ; 進料開爪位置有板
1757  LD      SM400  ; Run On\
      AND     L4642  ; 進料分流右側昇降上定點
      MEP
      AND     L2131  ; 分流前取框位置02進料側
      AND     L4636  ; 進料分流左側旋轉定點ON
      MOV     D1051 D1074  ; 進料分流右側框架尺寸    寬1=250
      DMOV    D1080 D1084  ; 進料分流左側框架尺寸    長0.000
      DMOV    K0 D1080
      MPS
      AND     D1065.0  ; 進料開爪位置有板
      SET     D1065.2  ; 進料分流右側有板
      MPP
      RST     D1065.0  ; 進料開爪位置有板
1774  LD      L4633  ; 進料分流左側昇降下定點
      MEP
      AND     L4630  ; 進料分流左側伸出定點
      AND     L4636  ; 進料分流左側旋轉定點ON
      MOV     D1073 D4001Z10
      MOV     K0 D1073
      MPS
      AND<    D4000 D1090  ; 左側爐內框數 / 爐內框架數量限制
      INC     D4000
      MOV     D4000 Z10
      MPP
      AND     D1065.1  ; 進料分流左側有板
      MOV     K1 D4051Z12
      RST     D1065.1  ; 進料分流左側有板
      AND<    D4050 D1091  ; 左側爐內板數 / 爐內板件數量限制
      INC     D4050
      MOV     D4050 Z12
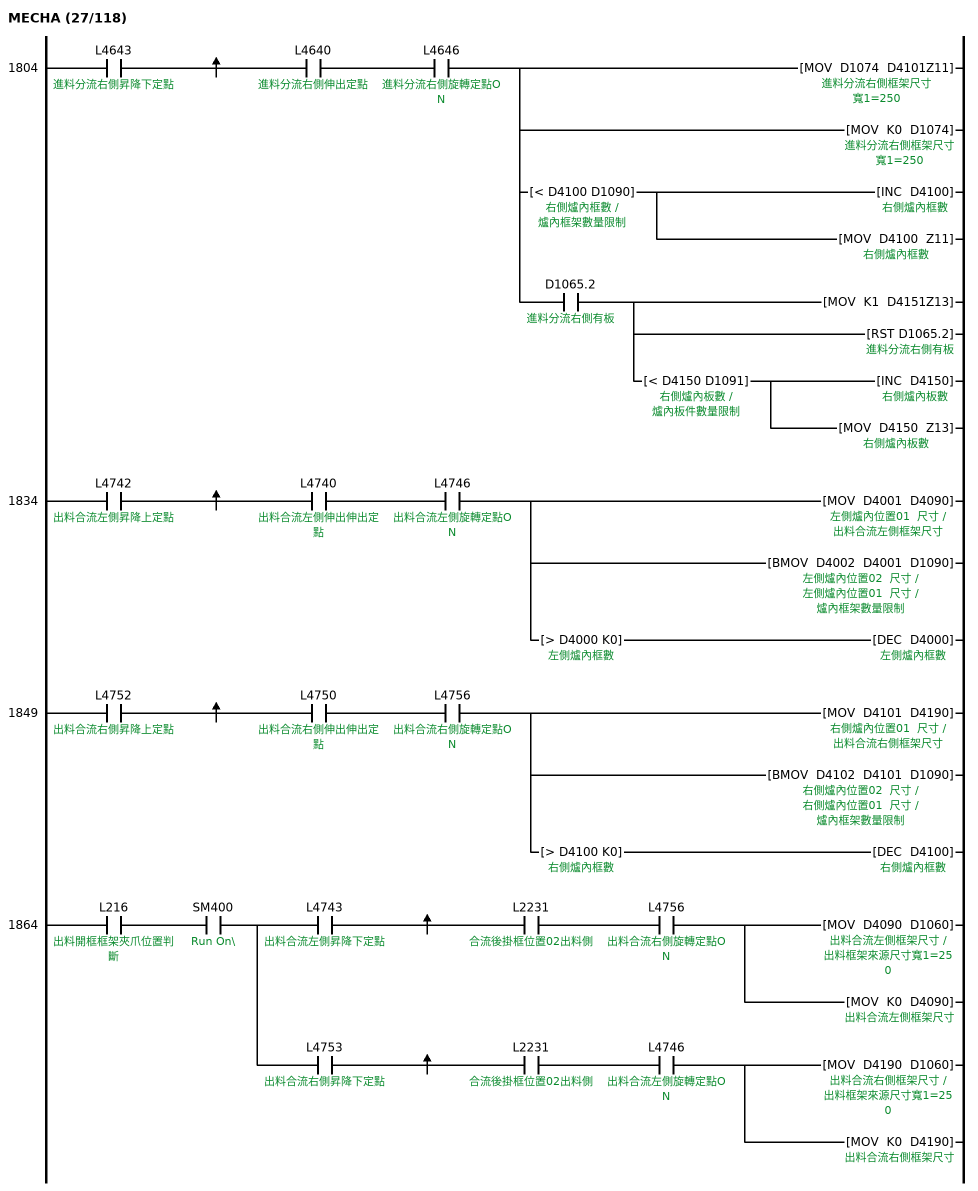
1804  LD      L4643  ; 進料分流右側昇降下定點
      MEP
      AND     L4640  ; 進料分流右側伸出定點
      AND     L4646  ; 進料分流右側旋轉定點ON
      MOV     D1074 D4101Z11
      MOV     K0 D1074
      MPS
      AND<    D4100 D1090  ; 右側爐內框數 / 爐內框架數量限制
      INC     D4100
      MOV     D4100 Z11
      MPP
      AND     D1065.2  ; 進料分流右側有板
      MOV     K1 D4151Z13
      RST     D1065.2  ; 進料分流右側有板
      AND<    D4150 D1091  ; 右側爐內板數 / 爐內板件數量限制
      INC     D4150
      MOV     D4150 Z13
1834  LD      L4742  ; 出料合流左側昇降上定點
      MEP
      AND     L4740  ; 出料合流左側伸出伸出定點
      AND     L4746  ; 出料合流左側旋轉定點ON
      MOV     D4001 D4090  ; 左側爐內位置01  尺寸 / 出料合流左側框架尺寸
      BMOV    D4002 D4001 D1090  ; 左側爐內位置02  尺寸
      AND>    D4000 K0  ; 左側爐內框數
      DEC     D4000
1849  LD      L4752  ; 出料合流右側昇降上定點
      MEP
      AND     L4750  ; 出料合流右側伸出伸出定點
      AND     L4756  ; 出料合流右側旋轉定點ON
      MOV     D4101 D4190  ; 右側爐內位置01  尺寸 / 出料合流右側框架尺寸
      BMOV    D4102 D4101 D1090  ; 右側爐內位置02  尺寸
      AND>    D4100 K0  ; 右側爐內框數
      DEC     D4100
1864  LD      L216  ; 出料開框框架夾爪位置判斷
      AND     SM400  ; Run On\
      MPS
      AND     L4743  ; 出料合流左側昇降下定點
      MEP
      AND     L2231  ; 合流後掛框位置02出料側
      AND     L4756  ; 出料合流右側旋轉定點ON
      MOV     D4090 D1060  ; 出料框架來源尺寸寬1=250
      MOV     K0 D4090
      MPP
      AND     L4753  ; 出料合流右側昇降下定點
      MEP
      AND     L2231  ; 合流後掛框位置02出料側
      AND     L4746  ; 出料合流左側旋轉定點ON
      MOV     D4190 D1060
      MOV     K0 D4190
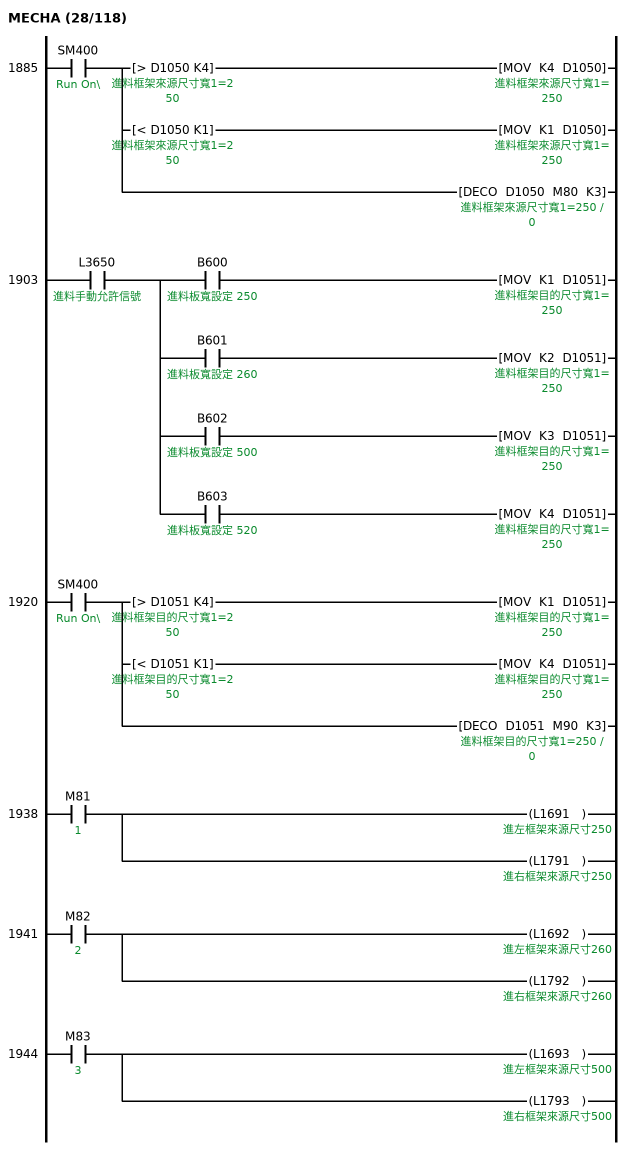
1885  LD      SM400  ; Run On\
      MPS
      AND>    D1050 K4  ; 進料框架來源尺寸寬1=250
      MOV     K4 D1050
      MRD
      AND<    D1050 K1  ; 進料框架來源尺寸寬1=250
      MOV     K1 D1050
      MPP
      DECO    D1050 M80 K3  ; 0
1903  LD      L3650  ; 進料手動允許信號
      MPS
      AND     B600  ; 進料板寬設定 250
      MOV     K1 D1051
      MRD
      AND     B601  ; 進料板寬設定 260
      MOV     K2 D1051
      MRD
      AND     B602  ; 進料板寬設定 500
      MOV     K3 D1051
      MPP
      AND     B603  ; 進料板寬設定 520
      MOV     K4 D1051
1920  LD      SM400  ; Run On\
      MPS
      AND>    D1051 K4  ; 進料框架目的尺寸寬1=250
      MOV     K1 D1051
      MRD
      AND<    D1051 K1  ; 進料框架目的尺寸寬1=250
      MOV     K4 D1051
      MPP
      DECO    D1051 M90 K3  ; 0
1938  LD      M81  ; 1
      OUT     L1691  ; 進左框架來源尺寸250
      OUT     L1791  ; 進右框架來源尺寸250
1941  LD      M82  ; 2
      OUT     L1692  ; 進左框架來源尺寸260
      OUT     L1792  ; 進右框架來源尺寸260
1944  LD      M83  ; 3
      OUT     L1693  ; 進左框架來源尺寸500
      OUT     L1793  ; 進右框架來源尺寸500
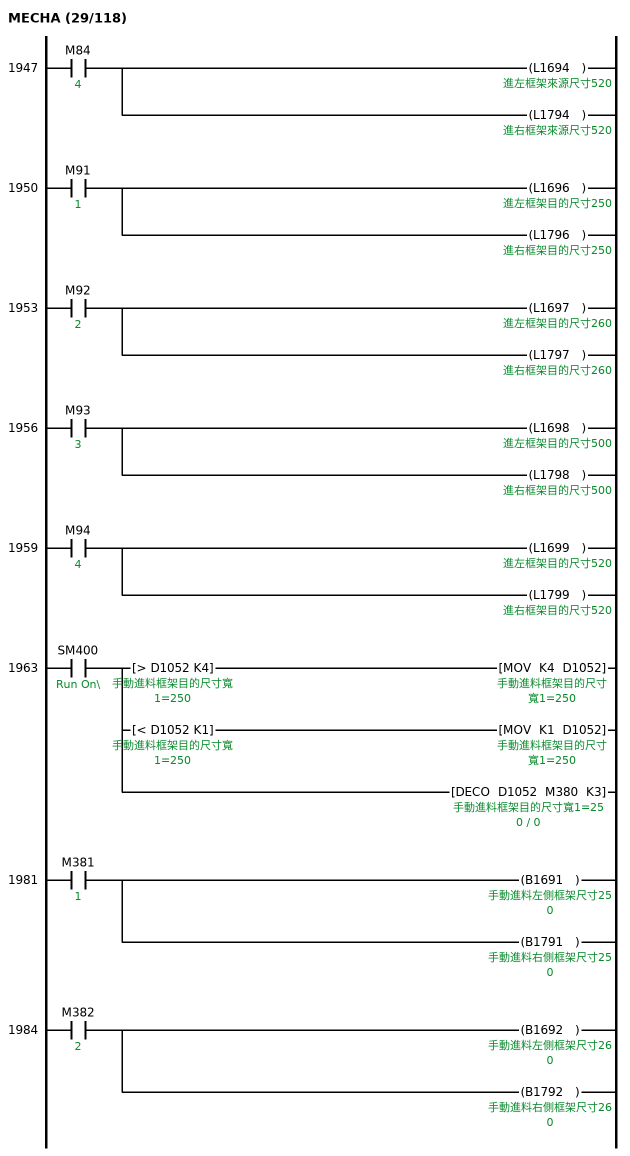
1947  LD      M84  ; 4
      OUT     L1694  ; 進左框架來源尺寸520
      OUT     L1794  ; 進右框架來源尺寸520
1950  LD      M91  ; 1
      OUT     L1696  ; 進左框架目的尺寸250
      OUT     L1796  ; 進右框架目的尺寸250
1953  LD      M92  ; 2
      OUT     L1697  ; 進左框架目的尺寸260
      OUT     L1797  ; 進右框架目的尺寸260
1956  LD      M93  ; 3
      OUT     L1698  ; 進左框架目的尺寸500
      OUT     L1798  ; 進右框架目的尺寸500
1959  LD      M94  ; 4
      OUT     L1699  ; 進左框架目的尺寸520
      OUT     L1799  ; 進右框架目的尺寸520
1963  LD      SM400  ; Run On\
      MPS
      AND>    D1052 K4  ; 手動進料框架目的尺寸寬1=250
      MOV     K4 D1052
      MRD
      AND<    D1052 K1  ; 手動進料框架目的尺寸寬1=250
      MOV     K1 D1052
      MPP
      DECO    D1052 M380 K3  ; 0
1981  LD      M381  ; 1
      OUT     B1691  ; 手動進料左側框架尺寸250
      OUT     B1791  ; 手動進料右側框架尺寸250
1984  LD      M382  ; 2
      OUT     B1692  ; 手動進料左側框架尺寸260
      OUT     B1792  ; 手動進料右側框架尺寸260
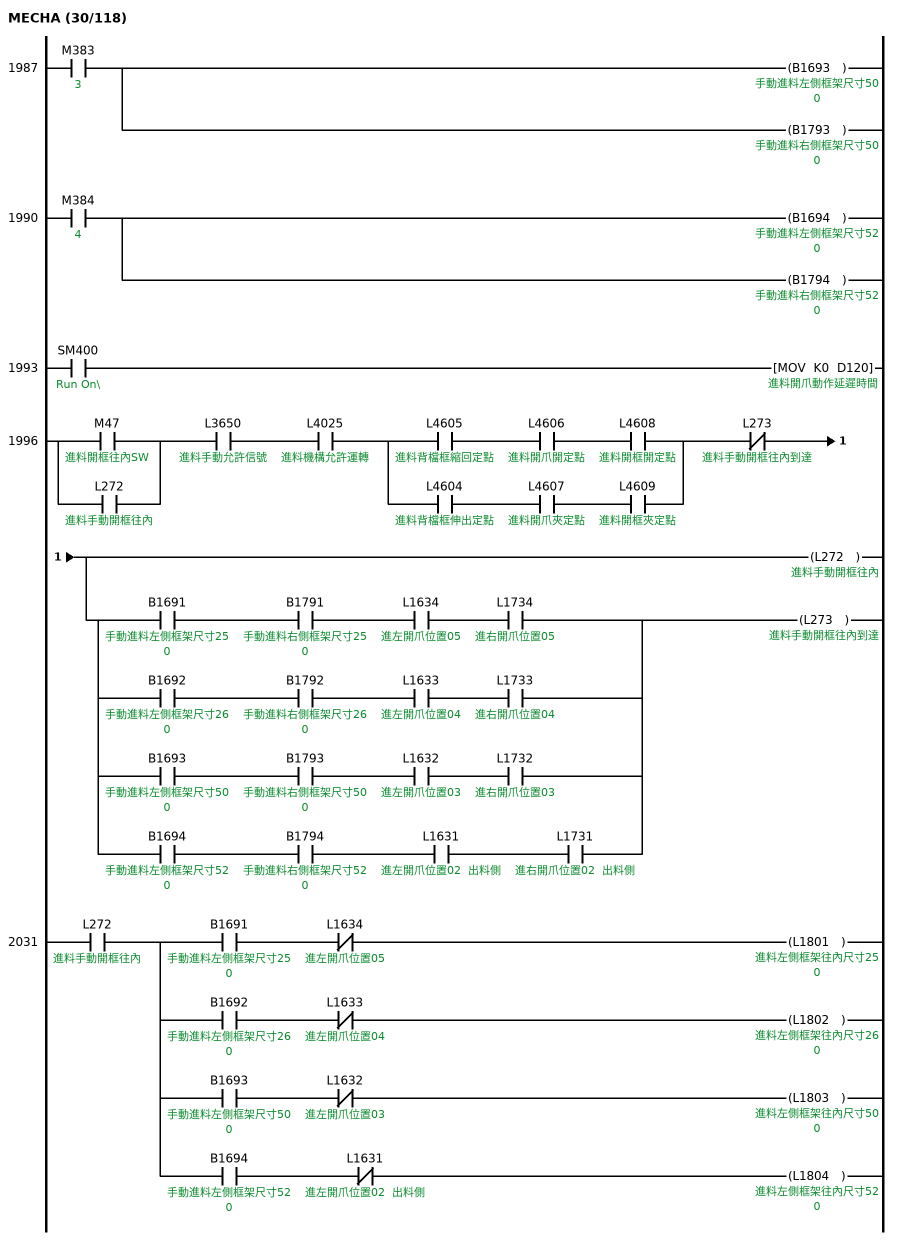
1987  LD      M383  ; 3
      OUT     B1693  ; 手動進料左側框架尺寸500
      OUT     B1793  ; 手動進料右側框架尺寸500
1990  LD      M384  ; 4
      OUT     B1694  ; 手動進料左側框架尺寸520
      OUT     B1794  ; 手動進料右側框架尺寸520
1993  LD      SM400  ; Run On\
      MOV     K0 D120  ; 進料開爪動作延遲時間
1996  LD      M47  ; 進料開框往內SW
      OR      L272  ; 進料手動開框往內
      AND     L3650  ; 進料手動允許信號
      AND     L4025  ; 進料機構允許運轉
      LD      L4605  ; 進料背檔框縮回定點
      AND     L4606  ; 進料開爪開定點
      AND     L4608  ; 進料開框開定點
      LD      L4604  ; 進料背檔框伸出定點
      AND     L4607  ; 進料開爪夾定點
      AND     L4609  ; 進料開框夾定點
      ORB
      ANB
      ANI     L273  ; 進料手動開框往內到達
      OUT     L272  ; 進料手動開框往內
      LD      B1691  ; 手動進料左側框架尺寸250
      AND     B1791  ; 手動進料右側框架尺寸250
      AND     L1634  ; 進左開爪位置05
      AND     L1734  ; 進右開爪位置05
      LD      B1692  ; 手動進料左側框架尺寸260
      AND     B1792  ; 手動進料右側框架尺寸260
      AND     L1633  ; 進左開爪位置04
      AND     L1733  ; 進右開爪位置04
      ORB
      LD      B1693  ; 手動進料左側框架尺寸500
      AND     B1793  ; 手動進料右側框架尺寸500
      AND     L1632  ; 進左開爪位置03
      AND     L1732  ; 進右開爪位置03
      ORB
      LD      B1694  ; 手動進料左側框架尺寸520
      AND     B1794  ; 手動進料右側框架尺寸520
      AND     L1631  ; 進左開爪位置02  出料側
      AND     L1731  ; 進右開爪位置02  出料側
      ORB
      ANB
      OUT     L273  ; 進料手動開框往內到達
2031  LD      L272  ; 進料手動開框往內
      MPS
      AND     B1691  ; 手動進料左側框架尺寸250
      ANI     L1634  ; 進左開爪位置05
      OUT     L1801  ; 進料左側框架往內尺寸250
      MRD
      AND     B1692  ; 手動進料左側框架尺寸260
      ANI     L1633  ; 進左開爪位置04
      OUT     L1802  ; 進料左側框架往內尺寸260
      MRD
      AND     B1693  ; 手動進料左側框架尺寸500
      ANI     L1632  ; 進左開爪位置03
      OUT     L1803  ; 進料左側框架往內尺寸500
      MPP
      AND     B1694  ; 手動進料左側框架尺寸520
      ANI     L1631  ; 進左開爪位置02  出料側
      OUT     L1804  ; 進料左側框架往內尺寸520
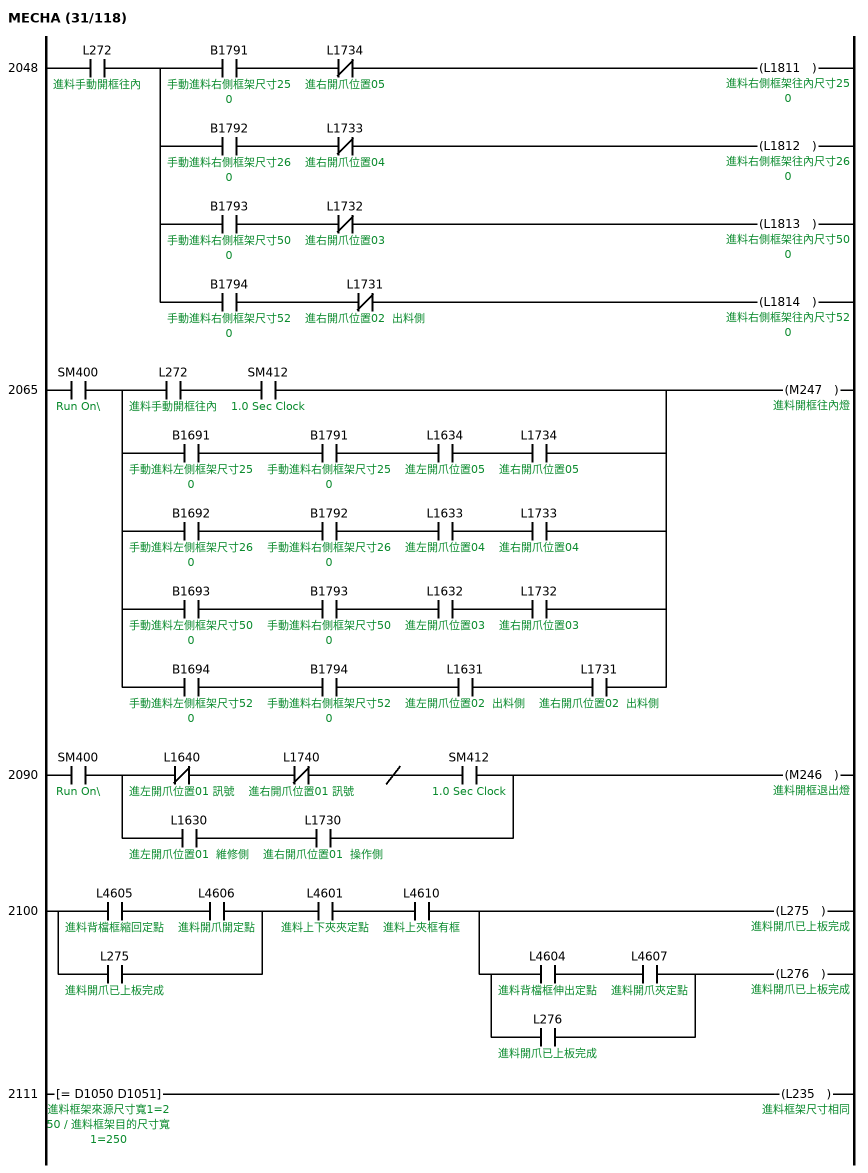
2048  LD      L272  ; 進料手動開框往內
      MPS
      AND     B1791  ; 手動進料右側框架尺寸250
      ANI     L1734  ; 進右開爪位置05
      OUT     L1811  ; 進料右側框架往內尺寸250
      MRD
      AND     B1792  ; 手動進料右側框架尺寸260
      ANI     L1733  ; 進右開爪位置04
      OUT     L1812  ; 進料右側框架往內尺寸260
      MRD
      AND     B1793  ; 手動進料右側框架尺寸500
      ANI     L1732  ; 進右開爪位置03
      OUT     L1813  ; 進料右側框架往內尺寸500
      MPP
      AND     B1794  ; 手動進料右側框架尺寸520
      ANI     L1731  ; 進右開爪位置02  出料側
      OUT     L1814  ; 進料右側框架往內尺寸520
2065  LD      SM400  ; Run On\
      LD      L272  ; 進料手動開框往內
      AND     SM412  ; 1.0 Sec Clock
      LD      B1691  ; 手動進料左側框架尺寸250
      AND     B1791  ; 手動進料右側框架尺寸250
      AND     L1634  ; 進左開爪位置05
      AND     L1734  ; 進右開爪位置05
      ORB
      LD      B1692  ; 手動進料左側框架尺寸260
      AND     B1792  ; 手動進料右側框架尺寸260
      AND     L1633  ; 進左開爪位置04
      AND     L1733  ; 進右開爪位置04
      ORB
      LD      B1693  ; 手動進料左側框架尺寸500
      AND     B1793  ; 手動進料右側框架尺寸500
      AND     L1632  ; 進左開爪位置03
      AND     L1732  ; 進右開爪位置03
      ORB
      LD      B1694  ; 手動進料左側框架尺寸520
      AND     B1794  ; 手動進料右側框架尺寸520
      AND     L1631  ; 進左開爪位置02  出料側
      AND     L1731  ; 進右開爪位置02  出料側
      ORB
      ANB
      OUT     M247  ; 進料開框往內燈
2090  LD      SM400  ; Run On\
      LDI     L1640  ; 進左開爪位置01 訊號
      ANI     L1740  ; 進右開爪位置01 訊號
      INV
      AND     SM412  ; 1.0 Sec Clock
      LD      L1630  ; 進左開爪位置01  維修側
      AND     L1730  ; 進右開爪位置01  操作側
      ORB
      ANB
      OUT     M246  ; 進料開框退出燈
2100  LD      L4605  ; 進料背檔框縮回定點
      AND     L4606  ; 進料開爪開定點
      OR      L275  ; 進料開爪已上板完成
      AND     L4601  ; 進料上下夾夾定點
      AND     L4610  ; 進料上夾框有框
      OUT     L275  ; 進料開爪已上板完成
      LD      L4604  ; 進料背檔框伸出定點
      AND     L4607  ; 進料開爪夾定點
      OR      L276  ; 進料開爪已上板完成
      ANB
      OUT     L276  ; 進料開爪已上板完成
2111  LD=     D1050 D1051  ; 進料框架來源尺寸寬1=250 / 進料框架目的尺寸寬1=250
      OUT     L235  ; 進料框架尺寸相同
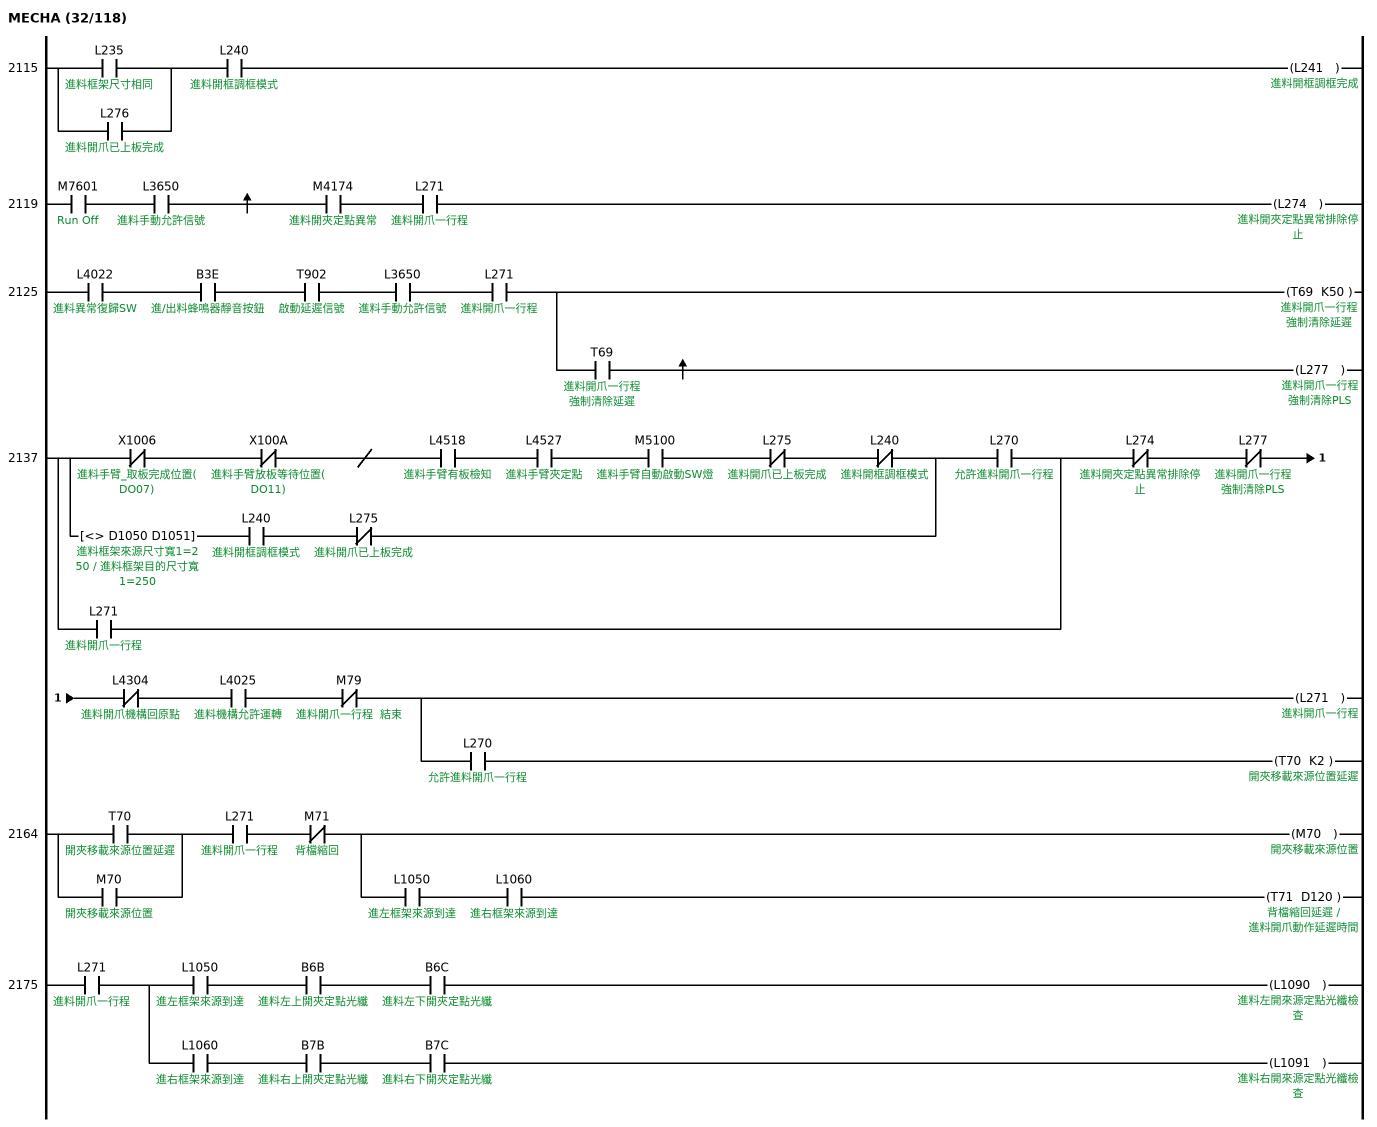
2115  LD      L235  ; 進料框架尺寸相同
      OR      L276  ; 進料開爪已上板完成
      AND     L240  ; 進料開框調框模式
      OUT     L241  ; 進料開框調框完成
2119  LD      M7601  ; Run Off
      AND     L3650  ; 進料手動允許信號
      MEP
      AND     M4174  ; 進料開夾定點異常
      AND     L271  ; 進料開爪一行程
      OUT     L274  ; 進料開夾定點異常排除停止
2125  LD      L4022  ; 進料異常復歸SW
      AND     B3E  ; 進/出料蜂鳴器靜音按鈕
      AND     T902  ; 啟動延遲信號
      AND     L3650  ; 進料手動允許信號
      AND     L271  ; 進料開爪一行程
      OUT     T69 K50  ; 進料開爪一行程  強制清除延遲
      AND     T69  ; 進料開爪一行程  強制清除延遲
      MEP
      OUT     L277  ; 進料開爪一行程  強制清除PLS
2137  LDI     X1006  ; 進料手臂_取板完成位置(DO07)
      ANI     X100A  ; 進料手臂放板等待位置(DO11)
      INV
      AND     L4518  ; 進料手臂有板檢知
      AND     L4527  ; 進料手臂夾定點
      AND     M5100  ; 進料手臂自動啟動SW燈
      ANI     L275  ; 進料開爪已上板完成
      ANI     L240  ; 進料開框調框模式
      LD<>    D1050 D1051  ; 進料框架來源尺寸寬1=250 / 進料框架目的尺寸寬1=250
      AND     L240  ; 進料開框調框模式
      ANI     L275  ; 進料開爪已上板完成
      ORB
      AND     L270  ; 允許進料開爪一行程
      OR      L271  ; 進料開爪一行程
      ANI     L274  ; 進料開夾定點異常排除停止
      ANI     L277  ; 進料開爪一行程  強制清除PLS
      ANI     L4304  ; 進料開爪機構回原點
      AND     L4025  ; 進料機構允許運轉
      ANI     M79  ; 進料開爪一行程  結束
      OUT     L271  ; 進料開爪一行程
      AND     L270  ; 允許進料開爪一行程
      OUT     T70 K2  ; 開夾移載來源位置延遲
2164  LD      T70  ; 開夾移載來源位置延遲
      OR      M70  ; 開夾移載來源位置
      AND     L271  ; 進料開爪一行程
      ANI     M71  ; 背檔縮回
      OUT     M70  ; 開夾移載來源位置
      AND     L1050  ; 進左框架來源到達
      AND     L1060  ; 進右框架來源到達
      OUT     T71 D120  ; 背檔縮回延遲 / 進料開爪動作延遲時間
2175  LD      L271  ; 進料開爪一行程
      MPS
      AND     L1050  ; 進左框架來源到達
      AND     B6B  ; 進料左上開夾定點光纖
      AND     B6C  ; 進料左下開夾定點光纖
      OUT     L1090  ; 進料左開來源定點光纖檢查
      MPP
      AND     L1060  ; 進右框架來源到達
      AND     B7B  ; 進料右上開夾定點光纖
      AND     B7C  ; 進料右下開夾定點光纖
      OUT     L1091  ; 進料右開來源定點光纖檢查
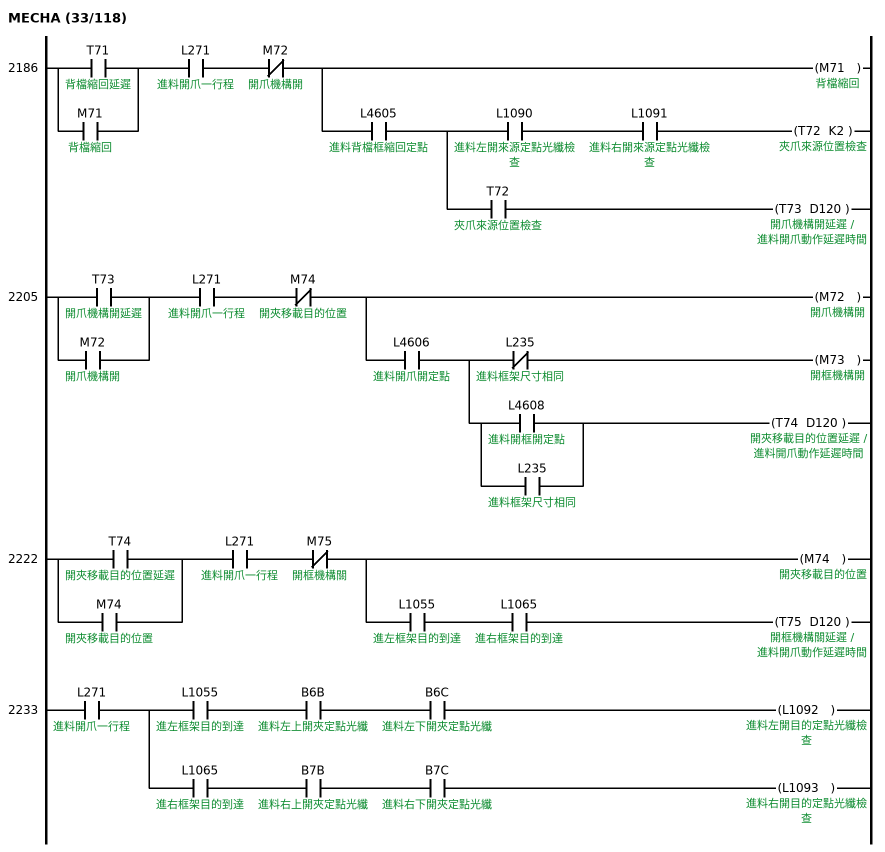
2186  LD      T71  ; 背檔縮回延遲
      OR      M71  ; 背檔縮回
      AND     L271  ; 進料開爪一行程
      ANI     M72  ; 開爪機構開
      OUT     M71  ; 背檔縮回
      AND     L4605  ; 進料背檔框縮回定點
      MPS
      AND     L1090  ; 進料左開來源定點光纖檢查
      AND     L1091  ; 進料右開來源定點光纖檢查
      OUT     T72 K2  ; 夾爪來源位置檢查
      MPP
      AND     T72  ; 夾爪來源位置檢查
      OUT     T73 D120  ; 開爪機構開延遲 / 進料開爪動作延遲時間
2205  LD      T73  ; 開爪機構開延遲
      OR      M72  ; 開爪機構開
      AND     L271  ; 進料開爪一行程
      ANI     M74  ; 開夾移載目的位置
      OUT     M72  ; 開爪機構開
      AND     L4606  ; 進料開爪開定點
      MPS
      ANI     L235  ; 進料框架尺寸相同
      OUT     M73  ; 開框機構開
      MPP
      LD      L4608  ; 進料開框開定點
      OR      L235  ; 進料框架尺寸相同
      ANB
      OUT     T74 D120  ; 開夾移載目的位置延遲 / 進料開爪動作延遲時間
2222  LD      T74  ; 開夾移載目的位置延遲
      OR      M74  ; 開夾移載目的位置
      AND     L271  ; 進料開爪一行程
      ANI     M75  ; 開框機構關
      OUT     M74  ; 開夾移載目的位置
      AND     L1055  ; 進左框架目的到達
      AND     L1065  ; 進右框架目的到達
      OUT     T75 D120  ; 開框機構關延遲 / 進料開爪動作延遲時間
2233  LD      L271  ; 進料開爪一行程
      MPS
      AND     L1055  ; 進左框架目的到達
      AND     B6B  ; 進料左上開夾定點光纖
      AND     B6C  ; 進料左下開夾定點光纖
      OUT     L1092  ; 進料左開目的定點光纖檢查
      MPP
      AND     L1065  ; 進右框架目的到達
      AND     B7B  ; 進料右上開夾定點光纖
      AND     B7C  ; 進料右下開夾定點光纖
      OUT     L1093  ; 進料右開目的定點光纖檢查
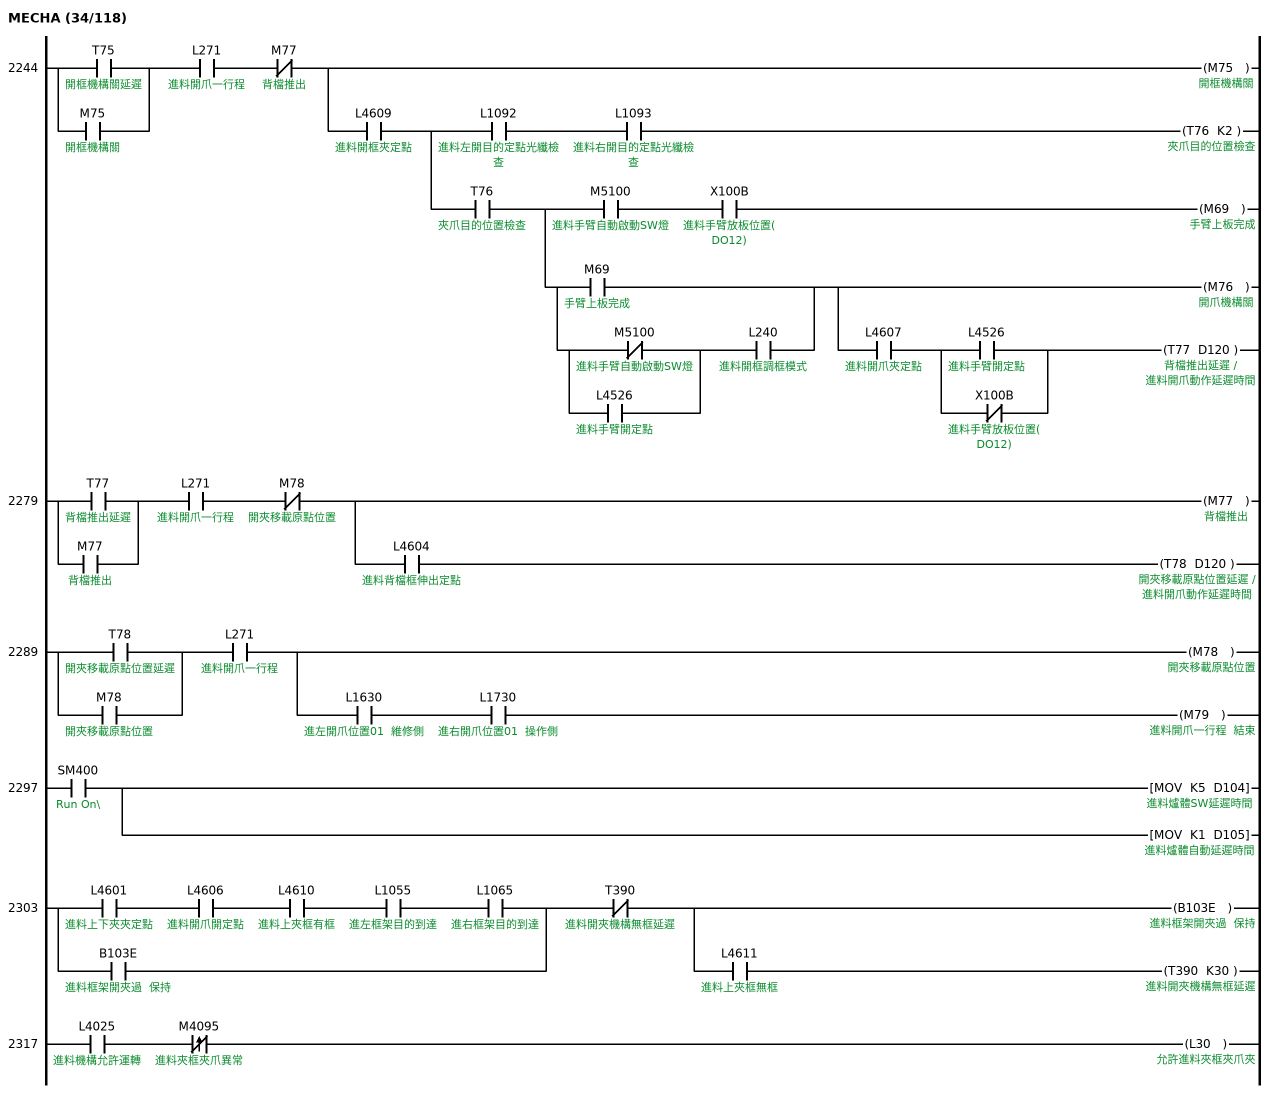
2244  LD      T75  ; 開框機構關延遲
      OR      M75  ; 開框機構關
      AND     L271  ; 進料開爪一行程
      ANI     M77  ; 背檔推出
      OUT     M75  ; 開框機構關
      AND     L4609  ; 進料開框夾定點
      MPS
      AND     L1092  ; 進料左開目的定點光纖檢查
      AND     L1093  ; 進料右開目的定點光纖檢查
      OUT     T76 K2  ; 夾爪目的位置檢查
      MPP
      AND     T76  ; 夾爪目的位置檢查
      MPS
      AND     M5100  ; 進料手臂自動啟動SW燈
      AND     X100B  ; 進料手臂放板位置(DO12)
      OUT     M69  ; 手臂上板完成
      MPP
      LD      M69  ; 手臂上板完成
      LDI     M5100  ; 進料手臂自動啟動SW燈
      OR      L4526  ; 進料手臂開定點
      AND     L240  ; 進料開框調框模式
      ORB
      ANB
      OUT     M76  ; 開爪機構關
      AND     L4607  ; 進料開爪夾定點
      LD      L4526  ; 進料手臂開定點
      ORI     X100B  ; 進料手臂放板位置(DO12)
      ANB
      OUT     T77 D120  ; 背檔推出延遲 / 進料開爪動作延遲時間
2279  LD      T77  ; 背檔推出延遲
      OR      M77  ; 背檔推出
      AND     L271  ; 進料開爪一行程
      ANI     M78  ; 開夾移載原點位置
      OUT     M77  ; 背檔推出
      AND     L4604  ; 進料背檔框伸出定點
      OUT     T78 D120  ; 開夾移載原點位置延遲 / 進料開爪動作延遲時間
2289  LD      T78  ; 開夾移載原點位置延遲
      OR      M78  ; 開夾移載原點位置
      AND     L271  ; 進料開爪一行程
      OUT     M78  ; 開夾移載原點位置
      AND     L1630  ; 進左開爪位置01  維修側
      AND     L1730  ; 進右開爪位置01  操作側
      OUT     M79  ; 進料開爪一行程  結束
2297  LD      SM400  ; Run On\
      MOV     K5 D104  ; 進料爐體SW延遲時間
      MOV     K1 D105  ; 進料爐體自動延遲時間
2303  LD      L4601  ; 進料上下夾夾定點
      AND     L4606  ; 進料開爪開定點
      AND     L4610  ; 進料上夾框有框
      AND     L1055  ; 進左框架目的到達
      AND     L1065  ; 進右框架目的到達
      OR      B103E  ; 進料框架開夾過  保持
      ANI     T390  ; 進料開夾機構無框延遲
      OUT     B103E  ; 進料框架開夾過  保持
      AND     L4611  ; 進料上夾框無框
      OUT     T390 K30  ; 進料開夾機構無框延遲
2317  LD      L4025  ; 進料機構允許運轉
      ANDPI   M4095  ; 進料夾框夾爪異常
      OUT     L30  ; 允許進料夾框夾爪夾
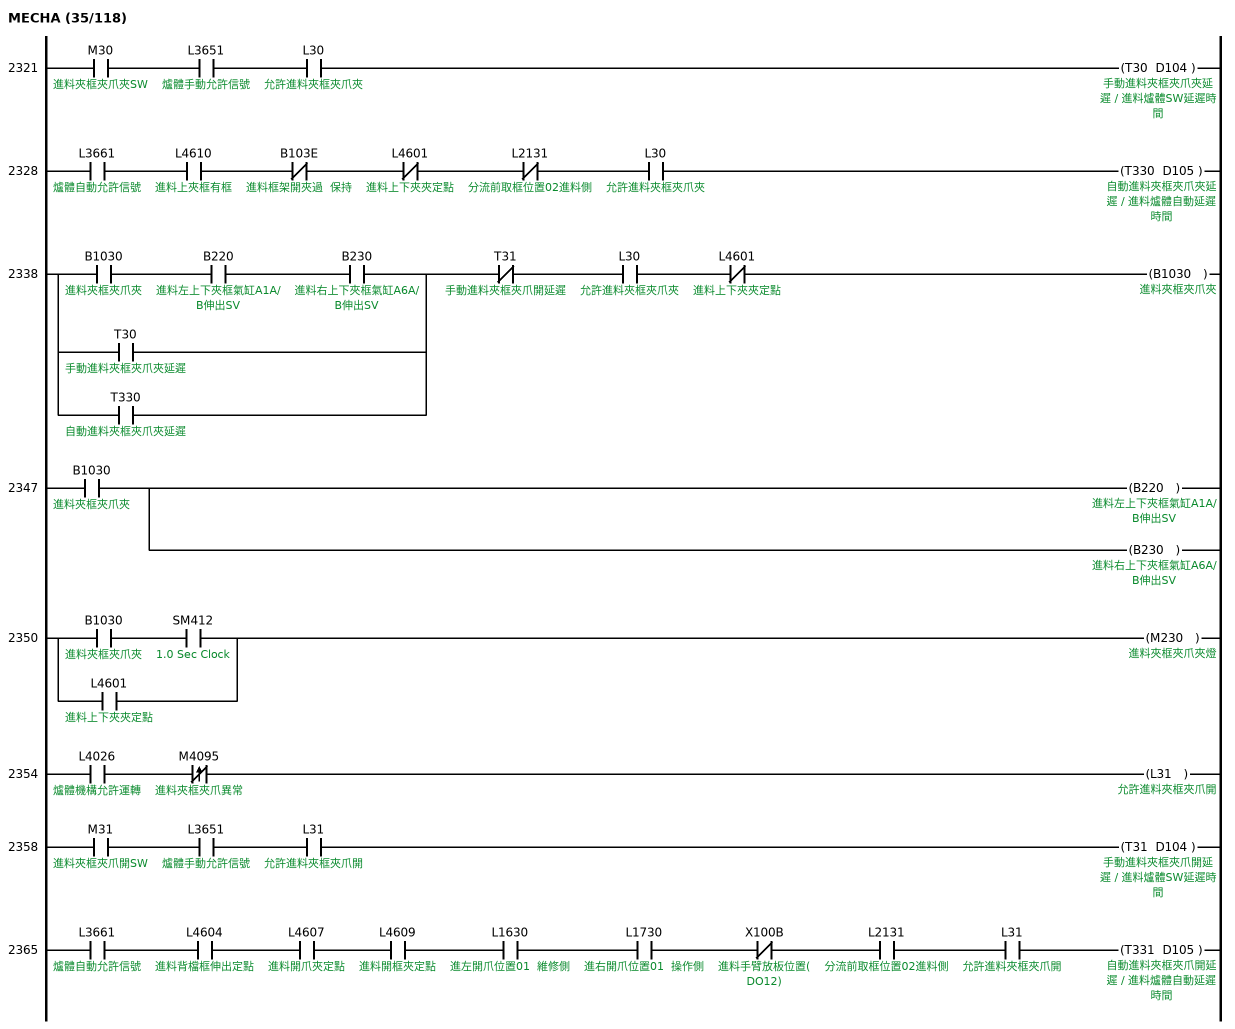
2321  LD      M30  ; 進料夾框夾爪夾SW
      AND     L3651  ; 爐體手動允許信號
      AND     L30  ; 允許進料夾框夾爪夾
      OUT     T30 D104  ; 手動進料夾框夾爪夾延遲 / 進料爐體SW延遲時間
2328  LD      L3661  ; 爐體自動允許信號
      AND     L4610  ; 進料上夾框有框
      ANI     B103E  ; 進料框架開夾過  保持
      ANI     L4601  ; 進料上下夾夾定點
      ANI     L2131  ; 分流前取框位置02進料側
      AND     L30  ; 允許進料夾框夾爪夾
      OUT     T330 D105  ; 自動進料夾框夾爪夾延遲 / 進料爐體自動延遲時間
2338  LD      B1030  ; 進料夾框夾爪夾
      AND     B220  ; 進料左上下夾框氣缸A1A/B伸出SV
      AND     B230  ; 進料右上下夾框氣缸A6A/B伸出SV
      OR      T30  ; 手動進料夾框夾爪夾延遲
      OR      T330  ; 自動進料夾框夾爪夾延遲
      ANI     T31  ; 手動進料夾框夾爪開延遲
      AND     L30  ; 允許進料夾框夾爪夾
      ANI     L4601  ; 進料上下夾夾定點
      OUT     B1030  ; 進料夾框夾爪夾
2347  LD      B1030  ; 進料夾框夾爪夾
      OUT     B220  ; 進料左上下夾框氣缸A1A/B伸出SV
      OUT     B230  ; 進料右上下夾框氣缸A6A/B伸出SV
2350  LD      B1030  ; 進料夾框夾爪夾
      AND     SM412  ; 1.0 Sec Clock
      OR      L4601  ; 進料上下夾夾定點
      OUT     M230  ; 進料夾框夾爪夾燈
2354  LD      L4026  ; 爐體機構允許運轉
      ANDPI   M4095  ; 進料夾框夾爪異常
      OUT     L31  ; 允許進料夾框夾爪開
2358  LD      M31  ; 進料夾框夾爪開SW
      AND     L3651  ; 爐體手動允許信號
      AND     L31  ; 允許進料夾框夾爪開
      OUT     T31 D104  ; 手動進料夾框夾爪開延遲 / 進料爐體SW延遲時間
2365  LD      L3661  ; 爐體自動允許信號
      AND     L4604  ; 進料背檔框伸出定點
      AND     L4607  ; 進料開爪夾定點
      AND     L4609  ; 進料開框夾定點
      AND     L1630  ; 進左開爪位置01  維修側
      AND     L1730  ; 進右開爪位置01  操作側
      ANI     X100B  ; 進料手臂放板位置(DO12)
      AND     L2131  ; 分流前取框位置02進料側
      AND     L31  ; 允許進料夾框夾爪開
      OUT     T331 D105  ; 自動進料夾框夾爪開延遲 / 進料爐體自動延遲時間
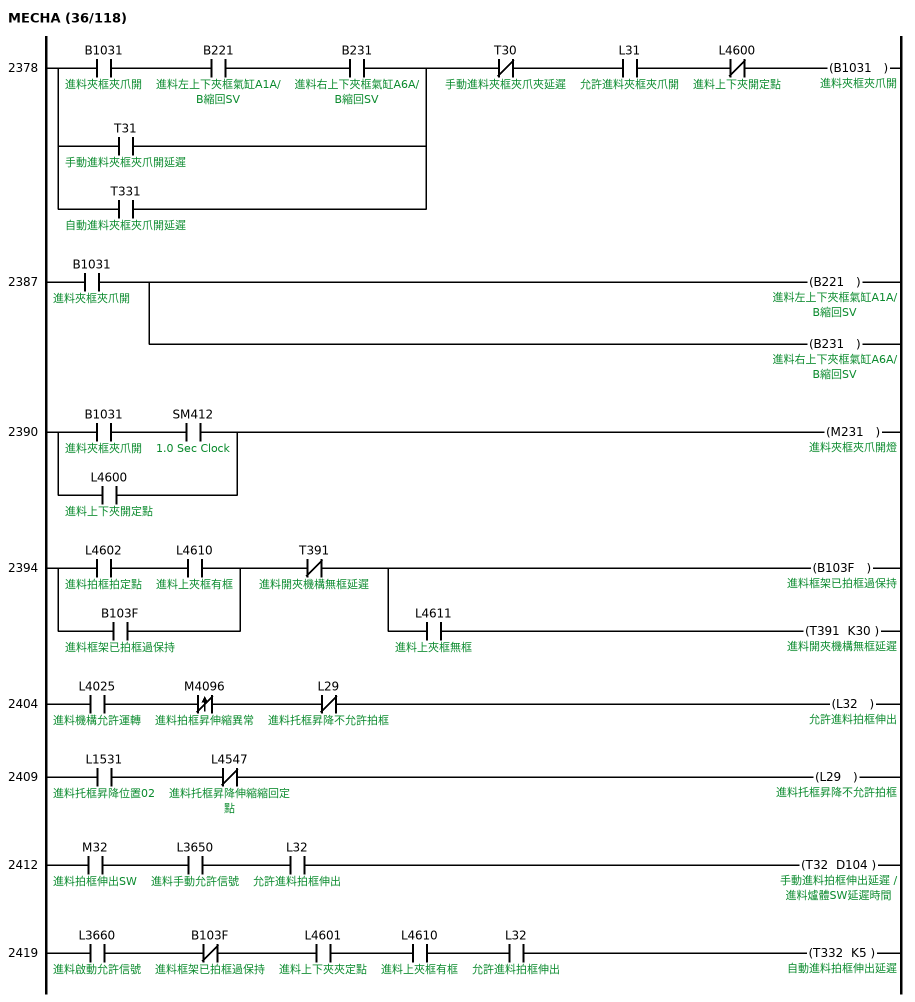
2378  LD      B1031  ; 進料夾框夾爪開
      AND     B221  ; 進料左上下夾框氣缸A1A/B縮回SV
      AND     B231  ; 進料右上下夾框氣缸A6A/B縮回SV
      OR      T31  ; 手動進料夾框夾爪開延遲
      OR      T331  ; 自動進料夾框夾爪開延遲
      ANI     T30  ; 手動進料夾框夾爪夾延遲
      AND     L31  ; 允許進料夾框夾爪開
      ANI     L4600  ; 進料上下夾開定點
      OUT     B1031  ; 進料夾框夾爪開
2387  LD      B1031  ; 進料夾框夾爪開
      OUT     B221  ; 進料左上下夾框氣缸A1A/B縮回SV
      OUT     B231  ; 進料右上下夾框氣缸A6A/B縮回SV
2390  LD      B1031  ; 進料夾框夾爪開
      AND     SM412  ; 1.0 Sec Clock
      OR      L4600  ; 進料上下夾開定點
      OUT     M231  ; 進料夾框夾爪開燈
2394  LD      L4602  ; 進料拍框拍定點
      AND     L4610  ; 進料上夾框有框
      OR      B103F  ; 進料框架已拍框過保持
      ANI     T391  ; 進料開夾機構無框延遲
      OUT     B103F  ; 進料框架已拍框過保持
      AND     L4611  ; 進料上夾框無框
      OUT     T391 K30  ; 進料開夾機構無框延遲
2404  LD      L4025  ; 進料機構允許運轉
      ANDPI   M4096  ; 進料拍框昇伸縮異常
      ANI     L29  ; 進料托框昇降不允許拍框
      OUT     L32  ; 允許進料拍框伸出
2409  LD      L1531  ; 進料托框昇降位置02
      ANI     L4547  ; 進料托框昇降伸縮縮回定點
      OUT     L29  ; 進料托框昇降不允許拍框
2412  LD      M32  ; 進料拍框伸出SW
      AND     L3650  ; 進料手動允許信號
      AND     L32  ; 允許進料拍框伸出
      OUT     T32 D104  ; 手動進料拍框伸出延遲 / 進料爐體SW延遲時間
2419  LD      L3660  ; 進料啟動允許信號
      ANI     B103F  ; 進料框架已拍框過保持
      AND     L4601  ; 進料上下夾夾定點
      AND     L4610  ; 進料上夾框有框
      AND     L32  ; 允許進料拍框伸出
      OUT     T332 K5  ; 自動進料拍框伸出延遲
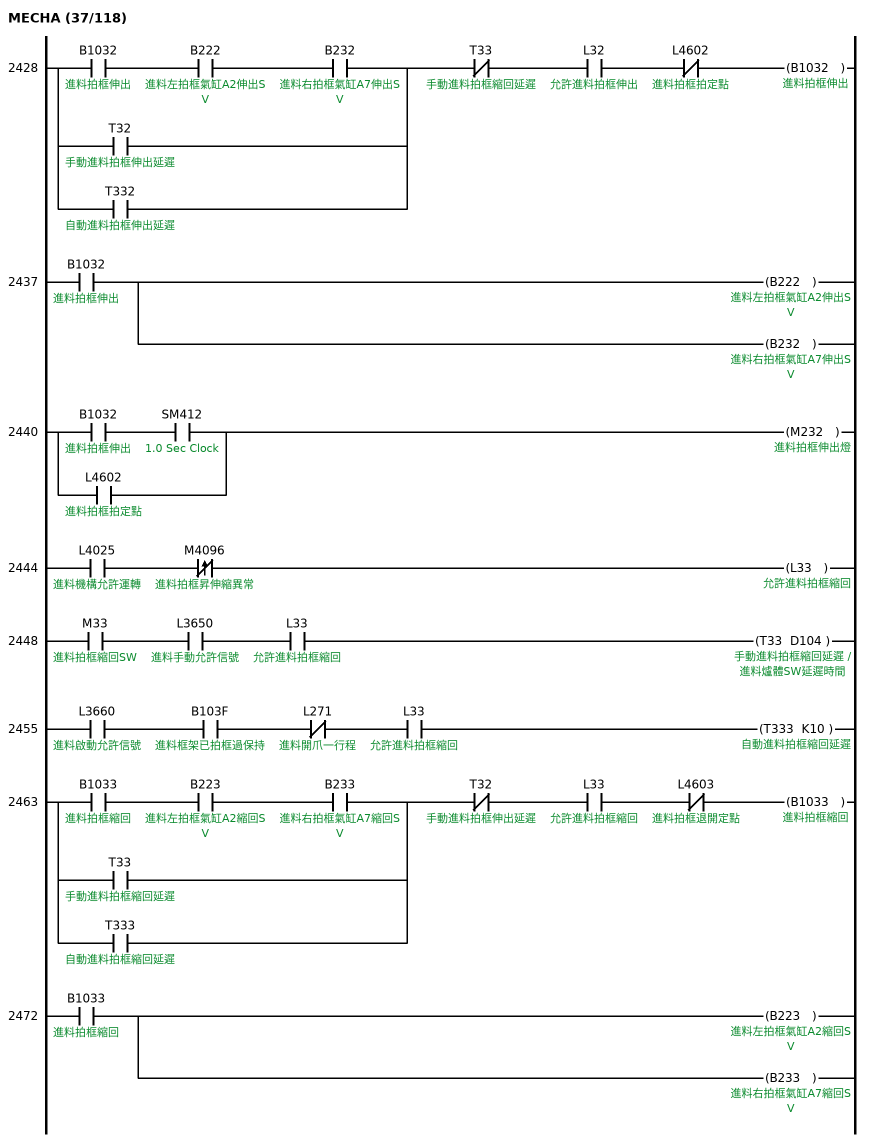
2428  LD      B1032  ; 進料拍框伸出
      AND     B222  ; 進料左拍框氣缸A2伸出SV
      AND     B232  ; 進料右拍框氣缸A7伸出SV
      OR      T32  ; 手動進料拍框伸出延遲
      OR      T332  ; 自動進料拍框伸出延遲
      ANI     T33  ; 手動進料拍框縮回延遲
      AND     L32  ; 允許進料拍框伸出
      ANI     L4602  ; 進料拍框拍定點
      OUT     B1032  ; 進料拍框伸出
2437  LD      B1032  ; 進料拍框伸出
      OUT     B222  ; 進料左拍框氣缸A2伸出SV
      OUT     B232  ; 進料右拍框氣缸A7伸出SV
2440  LD      B1032  ; 進料拍框伸出
      AND     SM412  ; 1.0 Sec Clock
      OR      L4602  ; 進料拍框拍定點
      OUT     M232  ; 進料拍框伸出燈
2444  LD      L4025  ; 進料機構允許運轉
      ANDPI   M4096  ; 進料拍框昇伸縮異常
      OUT     L33  ; 允許進料拍框縮回
2448  LD      M33  ; 進料拍框縮回SW
      AND     L3650  ; 進料手動允許信號
      AND     L33  ; 允許進料拍框縮回
      OUT     T33 D104  ; 手動進料拍框縮回延遲 / 進料爐體SW延遲時間
2455  LD      L3660  ; 進料啟動允許信號
      AND     B103F  ; 進料框架已拍框過保持
      ANI     L271  ; 進料開爪一行程
      AND     L33  ; 允許進料拍框縮回
      OUT     T333 K10  ; 自動進料拍框縮回延遲
2463  LD      B1033  ; 進料拍框縮回
      AND     B223  ; 進料左拍框氣缸A2縮回SV
      AND     B233  ; 進料右拍框氣缸A7縮回SV
      OR      T33  ; 手動進料拍框縮回延遲
      OR      T333  ; 自動進料拍框縮回延遲
      ANI     T32  ; 手動進料拍框伸出延遲
      AND     L33  ; 允許進料拍框縮回
      ANI     L4603  ; 進料拍框退開定點
      OUT     B1033  ; 進料拍框縮回
2472  LD      B1033  ; 進料拍框縮回
      OUT     B223  ; 進料左拍框氣缸A2縮回SV
      OUT     B233  ; 進料右拍框氣缸A7縮回SV
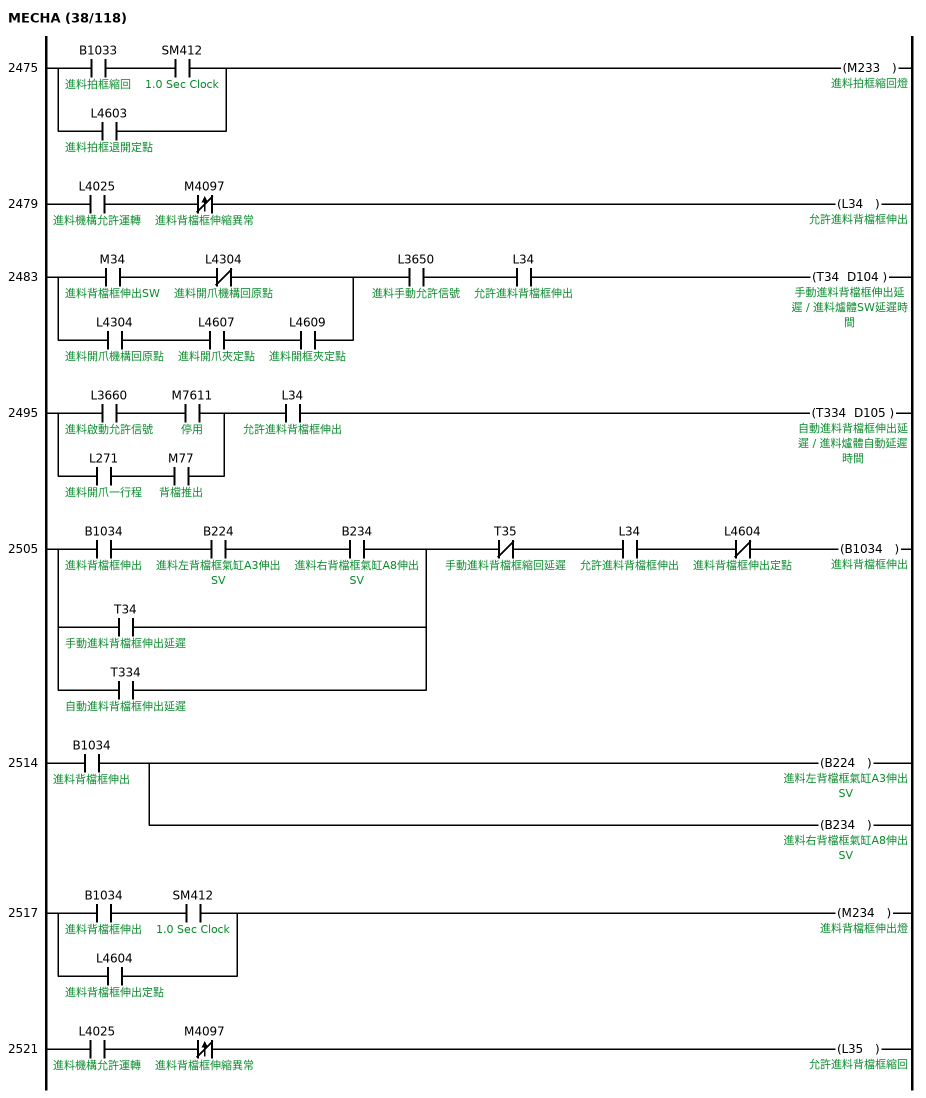
2475  LD      B1033  ; 進料拍框縮回
      AND     SM412  ; 1.0 Sec Clock
      OR      L4603  ; 進料拍框退開定點
      OUT     M233  ; 進料拍框縮回燈
2479  LD      L4025  ; 進料機構允許運轉
      ANDPI   M4097  ; 進料背檔框伸縮異常
      OUT     L34  ; 允許進料背檔框伸出
2483  LD      M34  ; 進料背檔框伸出SW
      ANI     L4304  ; 進料開爪機構回原點
      LD      L4304  ; 進料開爪機構回原點
      AND     L4607  ; 進料開爪夾定點
      AND     L4609  ; 進料開框夾定點
      ORB
      AND     L3650  ; 進料手動允許信號
      AND     L34  ; 允許進料背檔框伸出
      OUT     T34 D104  ; 手動進料背檔框伸出延遲 / 進料爐體SW延遲時間
2495  LD      L3660  ; 進料啟動允許信號
      AND     M7611  ; 停用
      LD      L271  ; 進料開爪一行程
      AND     M77  ; 背檔推出
      ORB
      AND     L34  ; 允許進料背檔框伸出
      OUT     T334 D105  ; 自動進料背檔框伸出延遲 / 進料爐體自動延遲時間
2505  LD      B1034  ; 進料背檔框伸出
      AND     B224  ; 進料左背檔框氣缸A3伸出SV
      AND     B234  ; 進料右背檔框氣缸A8伸出SV
      OR      T34  ; 手動進料背檔框伸出延遲
      OR      T334  ; 自動進料背檔框伸出延遲
      ANI     T35  ; 手動進料背檔框縮回延遲
      AND     L34  ; 允許進料背檔框伸出
      ANI     L4604  ; 進料背檔框伸出定點
      OUT     B1034  ; 進料背檔框伸出
2514  LD      B1034  ; 進料背檔框伸出
      OUT     B224  ; 進料左背檔框氣缸A3伸出SV
      OUT     B234  ; 進料右背檔框氣缸A8伸出SV
2517  LD      B1034  ; 進料背檔框伸出
      AND     SM412  ; 1.0 Sec Clock
      OR      L4604  ; 進料背檔框伸出定點
      OUT     M234  ; 進料背檔框伸出燈
2521  LD      L4025  ; 進料機構允許運轉
      ANDPI   M4097  ; 進料背檔框伸縮異常
      OUT     L35  ; 允許進料背檔框縮回
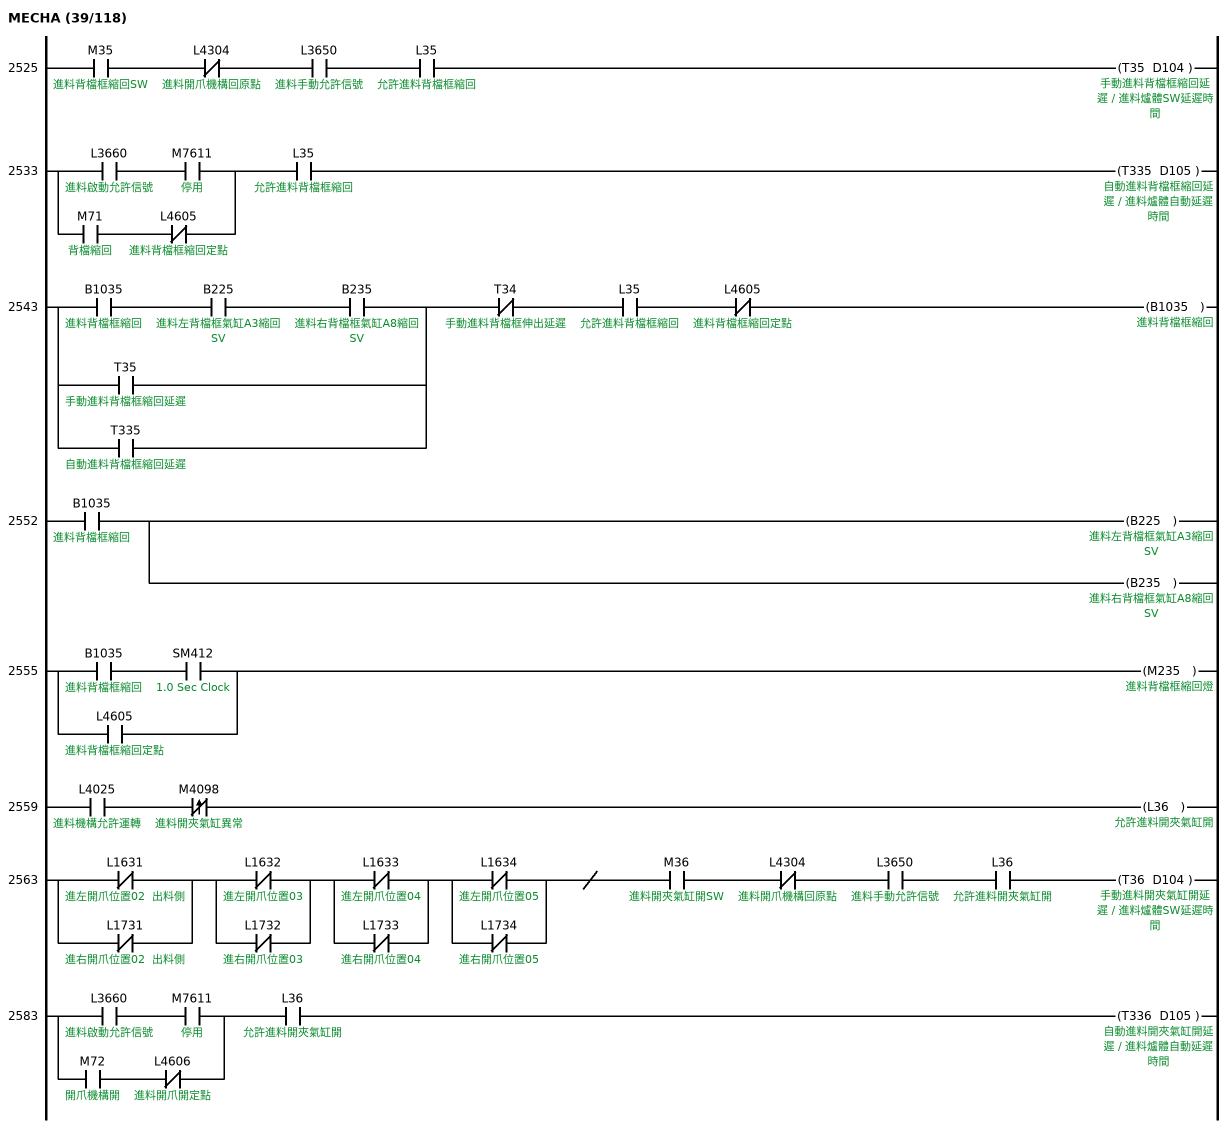
2525  LD      M35  ; 進料背檔框縮回SW
      ANI     L4304  ; 進料開爪機構回原點
      AND     L3650  ; 進料手動允許信號
      AND     L35  ; 允許進料背檔框縮回
      OUT     T35 D104  ; 手動進料背檔框縮回延遲 / 進料爐體SW延遲時間
2533  LD      L3660  ; 進料啟動允許信號
      AND     M7611  ; 停用
      LD      M71  ; 背檔縮回
      ANI     L4605  ; 進料背檔框縮回定點
      ORB
      AND     L35  ; 允許進料背檔框縮回
      OUT     T335 D105  ; 自動進料背檔框縮回延遲 / 進料爐體自動延遲時間
2543  LD      B1035  ; 進料背檔框縮回
      AND     B225  ; 進料左背檔框氣缸A3縮回SV
      AND     B235  ; 進料右背檔框氣缸A8縮回SV
      OR      T35  ; 手動進料背檔框縮回延遲
      OR      T335  ; 自動進料背檔框縮回延遲
      ANI     T34  ; 手動進料背檔框伸出延遲
      AND     L35  ; 允許進料背檔框縮回
      ANI     L4605  ; 進料背檔框縮回定點
      OUT     B1035  ; 進料背檔框縮回
2552  LD      B1035  ; 進料背檔框縮回
      OUT     B225  ; 進料左背檔框氣缸A3縮回SV
      OUT     B235  ; 進料右背檔框氣缸A8縮回SV
2555  LD      B1035  ; 進料背檔框縮回
      AND     SM412  ; 1.0 Sec Clock
      OR      L4605  ; 進料背檔框縮回定點
      OUT     M235  ; 進料背檔框縮回燈
2559  LD      L4025  ; 進料機構允許運轉
      ANDPI   M4098  ; 進料開夾氣缸異常
      OUT     L36  ; 允許進料開夾氣缸開
2563  LDI     L1631  ; 進左開爪位置02  出料側
      ORI     L1731  ; 進右開爪位置02  出料側
      LDI     L1632  ; 進左開爪位置03
      ORI     L1732  ; 進右開爪位置03
      ANB
      LDI     L1633  ; 進左開爪位置04
      ORI     L1733  ; 進右開爪位置04
      ANB
      LDI     L1634  ; 進左開爪位置05
      ORI     L1734  ; 進右開爪位置05
      ANB
      INV
      AND     M36  ; 進料開夾氣缸開SW
      ANI     L4304  ; 進料開爪機構回原點
      AND     L3650  ; 進料手動允許信號
      AND     L36  ; 允許進料開夾氣缸開
      OUT     T36 D104  ; 手動進料開夾氣缸開延遲 / 進料爐體SW延遲時間
2583  LD      L3660  ; 進料啟動允許信號
      AND     M7611  ; 停用
      LD      M72  ; 開爪機構開
      ANI     L4606  ; 進料開爪開定點
      ORB
      AND     L36  ; 允許進料開夾氣缸開
      OUT     T336 D105  ; 自動進料開夾氣缸開延遲 / 進料爐體自動延遲時間
